//     Term 29 (AT2000-0250)/CC Inputs/Current actual value Ch.12 <-> Data Pointer/CurrentActualValues[11]
//     Term 29 (AT2000-0250)/CC Inputs/Current actual value Ch.13 <-> Data Pointer/CurrentActualValues[12]
//     Term 29 (AT2000-0250)/CC Inputs/Current actual value Ch.14 <-> Data Pointer/CurrentActualValues[13]
//     Term 29 (AT2000-0250)/CC Inputs/Current actual value Ch.15 <-> Data Pointer/CurrentActualValues[14]
//     Term 29 (AT2000-0250)/CC Inputs/Current actual value Ch.2 <-> Data Pointer/CurrentActualValues[1]
//     Term 29 (AT2000-0250)/CC Inputs/Current actual value Ch.3 <-> Data Pointer/CurrentActualValues[2]
//     Term 29 (AT2000-0250)/CC Inputs/Current actual value Ch.4 <-> Data Pointer/CurrentActualValues[3]
//     Term 29 (AT2000-0250)/CC Inputs/Current actual value Ch.5 <-> Data Pointer/CurrentActualValues[4]
//     Term 29 (AT2000-0250)/CC Inputs/Current actual value Ch.6 <-> Data Pointer/CurrentActualValues[5]
//     Term 29 (AT2000-0250)/CC Inputs/Current actual value Ch.7 <-> Data Pointer/CurrentActualValues[6]
//     Term 29 (AT2000-0250)/CC Inputs/Current actual value Ch.8 <-> Data Pointer/CurrentActualValues[7]
//     Term 29 (AT2000-0250)/CC Inputs/Current actual value Ch.9 <-> Data Pointer/CurrentActualValues[8]
//     Term 29 (AT2000-0250)/CC Inputs/Status <-> Data Pointer/Status
//     Term 29 (AT2000-0250)/CC Outputs/Control <-> Data Pointer/Control
//     Term 29 (AT2000-0250)/CC Outputs/Current setpoint value Ch.1 <-> Data Pointer/CurrentSetpointValues[0]
//     Term 29 (AT2000-0250)/CC Outputs/Current setpoint value Ch.10 <-> Data Pointer/CurrentSetpointValues[9]
//     Term 29 (AT2000-0250)/CC Outputs/Current setpoint value Ch.11 <-> Data Pointer/CurrentSetpointValues[10]
//     Term 29 (AT2000-0250)/CC Outputs/Current setpoint value Ch.12 <-> Data Pointer/CurrentSetpointValues[11]
//     Term 29 (AT2000-0250)/CC Outputs/Current setpoint value Ch.13 <-> Data Pointer/CurrentSetpointValues[12]
//     Term 29 (AT2000-0250)/CC Outputs/Current setpoint value Ch.14 <-> Data Pointer/CurrentSetpointValues[13]
//     Term 29 (AT2000-0250)/CC Outputs/Current setpoint value Ch.15 <-> Data Pointer/CurrentSetpointValues[14]
//     Term 29 (AT2000-0250)/CC Outputs/Current setpoint value Ch.2 <-> Data Pointer/CurrentSetpointValues[1]
//     Term 29 (AT2000-0250)/CC Outputs/Current setpoint value Ch.3 <-> Data Pointer/CurrentSetpointValues[2]
//     Term 29 (AT2000-0250)/CC Outputs/Current setpoint value Ch.4 <-> Data Pointer/CurrentSetpointValues[3]
//     Term 29 (AT2000-0250)/CC Outputs/Current setpoint value Ch.5 <-> Data Pointer/CurrentSetpointValues[4]
//     Term 29 (AT2000-0250)/CC Outputs/Current setpoint value Ch.6 <-> Data Pointer/CurrentSetpointValues[5]
//     Term 29 (AT2000-0250)/CC Outputs/Current setpoint value Ch.7 <-> Data Pointer/CurrentSetpointValues[6]
//     Term 29 (AT2000-0250)/CC Outputs/Current setpoint value Ch.8 <-> Data Pointer/CurrentSetpointValues[7]
//     Term 29 (AT2000-0250)/CC Outputs/Current setpoint value Ch.9 <-> Data Pointer/CurrentSetpointValues[8]
//     Term 29 (AT2000-0250)/Term 30 (AT2000-5250)/FB Inputs/Value Channel 01 <-> Data Pointer/RawPositionValues[0]
//     Term 29 (AT2000-0250)/Term 30 (AT2000-5250)/FB Inputs/Value Channel 02 <-> Data Pointer/RawPositionValues[1]
//     Term 29 (AT2000-0250)/Term 30 (AT2000-5250)/FB Inputs/Value Channel 03 <-> Data Pointer/RawPositionValues[2]
//     Term 29 (AT2000-0250)/Term 30 (AT2000-5250)/FB Inputs/Value Channel 04 <-> Data Pointer/RawPositionValues[3]
//     Term 29 (AT2000-0250)/Term 30 (AT2000-5250)/FB Inputs/Value Channel 05 <-> Data Pointer/RawPositionValues[4]
//     Term 29 (AT2000-0250)/Term 30 (AT2000-5250)/FB Inputs/Value Channel 06 <-> Data Pointer/RawPositionValues[5]
//     Term 29 (AT2000-0250)/Term 30 (AT2000-5250)/FB Inputs/Value Channel 07 <-> Data Pointer/RawPositionValues[6]
//     Term 29 (AT2000-0250)/Term 30 (AT2000-5250)/FB Inputs/Value Channel 08 <-> Data Pointer/RawPositionValues[7]
//     Term 29 (AT2000-0250)/Term 30 (AT2000-5250)/FB Inputs/Value Channel 09 <-> Data Pointer/RawPositionValues[8]
//     Term 29 (AT2000-0250)/Term 30 (AT2000-5250)/FB Inputs/Value Channel 10 <-> Data Pointer/RawPositionValues[9]
//     Term 29 (AT2000-0250)/Term 30 (AT2000-5250)/FB Inputs/Value Channel 11 <-> Data Pointer/RawPositionValues[10]
//     Term 29 (AT2000-0250)/Term 30 (AT2000-5250)/FB Inputs/Value Channel 12 <-> Data Pointer/RawPositionValues[11]
//     Term 29 (AT2000-0250)/Term 30 (AT2000-5250)/FB Inputs/Value Channel 13 <-> Data Pointer/RawPositionValues[12]
//     Term 29 (AT2000-0250)/Term 30 (AT2000-5250)/FB Inputs/Value Channel 14 <-> Data Pointer/RawPositionValues[13]
//     Term 29 (AT2000-0250)/Term 30 (AT2000-5250)/FB Inputs/Value Channel 15 <-> Data Pointer/RawPositionValues[14]
//     Term 29 (AT2000-0250)/Term 30 (AT2000-5250)/FB Inputs/Value Channel 16 <-> Data Pointer/RawPositionValues[15]
//     Term 29 (AT2000-0250)/Term 30 (AT2000-5250)/FB Inputs/Value Channel 17 <-> Data Pointer/RawPositionValues[16]
//     Term 29 (AT2000-0250)/Term 30 (AT2000-5250)/FB Inputs/Value Channel 18 <-> Data Pointer/RawPositionValues[17]
//     Term 29 (AT2000-0250)/Term 30 (AT2000-5250)/FB Inputs/Value Channel 19 <-> Data Pointer/RawPositionValues[18]
//     Term 29 (AT2000-0250)/Term 30 (AT2000-5250)/FB Inputs/Value Channel 20 <-> Data Pointer/RawPositionValues[19]
//     Term 29 (AT2000-0250)/Term 30 (AT2000-5250)/FB Inputs/Value Channel 21 <-> Data Pointer/RawPositionValues[20]
//     Term 29 (AT2000-0250)/Term 30 (AT2000-5250)/FB Inputs/Value Channel 22 <-> Data Pointer/RawPositionValues[21]
//     Term 29 (AT2000-0250)/Term 30 (AT2000-5250)/FB Inputs/Value Channel 23 <-> Data Pointer/RawPositionValues[22]
//     Term 29 (AT2000-0250)/Term 30 (AT2000-5250)/FB Inputs/Value Channel 24 <-> Data Pointer/RawPositionValues[23]
//     Term 29 (AT2000-0250)/Term 30 (AT2000-5250)/FB Inputs/Value Channel 25 <-> Data Pointer/RawPositionValues[24]
//     Term 29 (AT2000-0250)/Term 30 (AT2000-5250)/FB Inputs/Value Channel 26 <-> Data Pointer/RawPositionValues[25]
//     Term 29 (AT2000-0250)/Term 30 (AT2000-5250)/FB Inputs/Value Channel 27 <-> Data Pointer/RawPositionValues[26]
//     Term 29 (AT2000-0250)/Term 30 (AT2000-5250)/FB Inputs/Value Channel 28 <-> Data Pointer/RawPositionValues[27]
//     Term 29 (AT2000-0250)/Term 30 (AT2000-5250)/FB Inputs/Value Channel 29 <-> Data Pointer/RawPositionValues[28]
//     Term 29 (AT2000-0250)/Term 30 (AT2000-5250)/FB Inputs/Value Channel 30 <-> Data Pointer/RawPositionValues[29]
//     Term 29 (AT2000-0250)/Term 30 (AT2000-5250)/FB Inputs/Value Channel 31 <-> Data Pointer/RawPositionValues[30]
//     Term 29 (AT2000-0250)/Term 30 (AT2000-5250)/FB Inputs/Value Channel 32 <-> Data Pointer/RawPositionValues[31]
//   Device 4 (EtherCAT) <-> TcCOM Objects/Object7 (CTcIoXtsDrv)/XTS Module Adapter_Obj15 (AT2050_X500)
//     Term 31 (AT2050-0500)/CC Inputs/Current actual value Ch.1 <-> Data Pointer/CurrentActualValues[0]
//     Term 31 (AT2050-0500)/CC Inputs/Current actual value Ch.10 <-> Data Pointer/CurrentActualValues[9]
//     Term 31 (AT2050-0500)/CC Inputs/Current actual value Ch.11 <-> Data Pointer/CurrentActualValues[10]
//     Term 31 (AT2050-0500)/CC Inputs/Current actual value Ch.12 <-> Data Pointer/CurrentActualValues[11]
//     Term 31 (AT2050-0500)/CC Inputs/Current actual value Ch.13 <-> Data Pointer/CurrentActualValues[12]
//     Term 31 (AT2050-0500)/CC Inputs/Current actual value Ch.14 <-> Data Pointer/CurrentActualValues[13]
//     Term 31 (AT2050-0500)/CC Inputs/Current actual value Ch.15 <-> Data Pointer/CurrentActualValues[14]
//     Term 31 (AT2050-0500)/CC Inputs/Current actual value Ch.2 <-> Data Pointer/CurrentActualValues[1]
//     Term 31 (AT2050-0500)/CC Inputs/Current actual value Ch.3 <-> Data Pointer/CurrentActualValues[2]
//     Term 31 (AT2050-0500)/CC Inputs/Current actual value Ch.4 <-> Data Pointer/CurrentActualValues[3]
//     Term 31 (AT2050-0500)/CC Inputs/Current actual value Ch.5 <-> Data Pointer/CurrentActualValues[4]
//     Term 31 (AT2050-0500)/CC Inputs/Current actual value Ch.6 <-> Data Pointer/CurrentActualValues[5]
//     Term 31 (AT2050-0500)/CC Inputs/Current actual value Ch.7 <-> Data Pointer/CurrentActualValues[6]
//     Term 31 (AT2050-0500)/CC Inputs/Current actual value Ch.8 <-> Data Pointer/CurrentActualValues[7]
//     Term 31 (AT2050-0500)/CC Inputs/Current actual value Ch.9 <-> Data Pointer/CurrentActualValues[8]
//     Term 31 (AT2050-0500)/CC Inputs/Status <-> Data Pointer/Status
//     Term 31 (AT2050-0500)/CC Outputs/Control <-> Data Pointer/Control
//     Term 31 (AT2050-0500)/CC Outputs/Current setpoint value Ch.1 <-> Data Pointer/CurrentSetpointValues[0]
//     Term 31 (AT2050-0500)/CC Outputs/Current setpoint value Ch.10 <-> Data Pointer/CurrentSetpointValues[9]
//     Term 31 (AT2050-0500)/CC Outputs/Current setpoint value Ch.11 <-> Data Pointer/CurrentSetpointValues[10]
//     Term 31 (AT2050-0500)/CC Outputs/Current setpoint value Ch.12 <-> Data Pointer/CurrentSetpointValues[11]
//     Term 31 (AT2050-0500)/CC Outputs/Current setpoint value Ch.13 <-> Data Pointer/CurrentSetpointValues[12]
//     Term 31 (AT2050-0500)/CC Outputs/Current setpoint value Ch.14 <-> Data Pointer/CurrentSetpointValues[13]
//     Term 31 (AT2050-0500)/CC Outputs/Current setpoint value Ch.15 <-> Data Pointer/CurrentSetpointValues[14]
//     Term 31 (AT2050-0500)/CC Outputs/Current setpoint value Ch.2 <-> Data Pointer/CurrentSetpointValues[1]
//     Term 31 (AT2050-0500)/CC Outputs/Current setpoint value Ch.3 <-> Data Pointer/CurrentSetpointValues[2]
//     Term 31 (AT2050-0500)/CC Outputs/Current setpoint value Ch.4 <-> Data Pointer/CurrentSetpointValues[3]
//     Term 31 (AT2050-0500)/CC Outputs/Current setpoint value Ch.5 <-> Data Pointer/CurrentSetpointValues[4]
//     Term 31 (AT2050-0500)/CC Outputs/Current setpoint value Ch.6 <-> Data Pointer/CurrentSetpointValues[5]
//     Term 31 (AT2050-0500)/CC Outputs/Current setpoint value Ch.7 <-> Data Pointer/CurrentSetpointValues[6]
//     Term 31 (AT2050-0500)/CC Outputs/Current setpoint value Ch.8 <-> Data Pointer/CurrentSetpointValues[7]
//     Term 31 (AT2050-0500)/CC Outputs/Current setpoint value Ch.9 <-> Data Pointer/CurrentSetpointValues[8]
//     Term 31 (AT2050-0500)/Term 32 (AT2050-5500)/FB Inputs/Value Channel 01 <-> Data Pointer/RawPositionValues[0]
//     Term 31 (AT2050-0500)/Term 32 (AT2050-5500)/FB Inputs/Value Channel 02 <-> Data Pointer/RawPositionValues[1]
//     Term 31 (AT2050-0500)/Term 32 (AT2050-5500)/FB Inputs/Value Channel 03 <-> Data Pointer/RawPositionValues[2]
//     Term 31 (AT2050-0500)/Term 32 (AT2050-5500)/FB Inputs/Value Channel 04 <-> Data Pointer/RawPositionValues[3]
//     Term 31 (AT2050-0500)/Term 32 (AT2050-5500)/FB Inputs/Value Channel 05 <-> Data Pointer/RawPositionValues[4]
//     Term 31 (AT2050-0500)/Term 32 (AT2050-5500)/FB Inputs/Value Channel 06 <-> Data Pointer/RawPositionValues[5]
//     Term 31 (AT2050-0500)/Term 32 (AT2050-5500)/FB Inputs/Value Channel 07 <-> Data Pointer/RawPositionValues[6]
//     Term 31 (AT2050-0500)/Term 32 (AT2050-5500)/FB Inputs/Value Channel 08 <-> Data Pointer/RawPositionValues[7]
//     Term 31 (AT2050-0500)/Term 32 (AT2050-5500)/FB Inputs/Value Channel 09 <-> Data Pointer/RawPositionValues[8]
//     Term 31 (AT2050-0500)/Term 32 (AT2050-5500)/FB Inputs/Value Channel 10 <-> Data Pointer/RawPositionValues[9]
//     Term 31 (AT2050-0500)/Term 32 (AT2050-5500)/FB Inputs/Value Channel 11 <-> Data Pointer/RawPositionValues[10]
//     Term 31 (AT2050-0500)/Term 32 (AT2050-5500)/FB Inputs/Value Channel 12 <-> Data Pointer/RawPositionValues[11]
//     Term 31 (AT2050-0500)/Term 32 (AT2050-5500)/FB Inputs/Value Channel 13 <-> Data Pointer/RawPositionValues[12]
//     Term 31 (AT2050-0500)/Term 32 (AT2050-5500)/FB Inputs/Value Channel 14 <-> Data Pointer/RawPositionValues[13]
//     Term 31 (AT2050-0500)/Term 32 (AT2050-5500)/FB Inputs/Value Channel 15 <-> Data Pointer/RawPositionValues[14]
//     Term 31 (AT2050-0500)/Term 32 (AT2050-5500)/FB Inputs/Value Channel 16 <-> Data Pointer/RawPositionValues[15]
//     Term 31 (AT2050-0500)/Term 32 (AT2050-5500)/FB Inputs/Value Channel 17 <-> Data Pointer/RawPositionValues[16]
//     Term 31 (AT2050-0500)/Term 32 (AT2050-5500)/FB Inputs/Value Channel 18 <-> Data Pointer/RawPositionValues[17]
//     Term 31 (AT2050-0500)/Term 32 (AT2050-5500)/FB Inputs/Value Channel 19 <-> Data Pointer/RawPositionValues[18]
//     Term 31 (AT2050-0500)/Term 32 (AT2050-5500)/FB Inputs/Value Channel 20 <-> Data Pointer/RawPositionValues[19]
//     Term 31 (AT2050-0500)/Term 32 (AT2050-5500)/FB Inputs/Value Channel 21 <-> Data Pointer/RawPositionValues[20]
//     Term 31 (AT2050-0500)/Term 32 (AT2050-5500)/FB Inputs/Value Channel 22 <-> Data Pointer/RawPositionValues[21]
//     Term 31 (AT2050-0500)/Term 32 (AT2050-5500)/FB Inputs/Value Channel 23 <-> Data Pointer/RawPositionValues[22]
//     Term 31 (AT2050-0500)/Term 32 (AT2050-5500)/FB Inputs/Value Channel 24 <-> Data Pointer/RawPositionValues[23]
//     Term 31 (AT2050-0500)/Term 32 (AT2050-5500)/FB Inputs/Value Channel 25 <-> Data Pointer/RawPositionValues[24]
//     Term 31 (AT2050-0500)/Term 32 (AT2050-5500)/FB Inputs/Value Channel 26 <-> Data Pointer/RawPositionValues[25]
//     Term 31 (AT2050-0500)/Term 32 (AT2050-5500)/FB Inputs/Value Channel 27 <-> Data Pointer/RawPositionValues[26]
//     Term 31 (AT2050-0500)/Term 32 (AT2050-5500)/FB Inputs/Value Channel 28 <-> Data Pointer/RawPositionValues[27]
//     Term 31 (AT2050-0500)/Term 32 (AT2050-5500)/FB Inputs/Value Channel 29 <-> Data Pointer/RawPositionValues[28]
//     Term 31 (AT2050-0500)/Term 32 (AT2050-5500)/FB Inputs/Value Channel 30 <-> Data Pointer/RawPositionValues[29]
//     Term 31 (AT2050-0500)/Term 32 (AT2050-5500)/FB Inputs/Value Channel 31 <-> Data Pointer/RawPositionValues[30]
//     Term 31 (AT2050-0500)/Term 32 (AT2050-5500)/FB Inputs/Value Channel 32 <-> Data Pointer/RawPositionValues[31]
//   Device 4 (EtherCAT) <-> TcCOM Objects/Object7 (CTcIoXtsDrv)/XTS Module Adapter_Obj16 (AT2050_X501)
//     Term 33 (AT2050-0501)/CC Inputs/Current actual value Ch.1 <-> Data Pointer/CurrentActualValues[0]
//     Term 33 (AT2050-0501)/CC Inputs/Current actual value Ch.10 <-> Data Pointer/CurrentActualValues[9]
//     Term 33 (AT2050-0501)/CC Inputs/Current actual value Ch.11 <-> Data Pointer/CurrentActualValues[10]
//     Term 33 (AT2050-0501)/CC Inputs/Current actual value Ch.12 <-> Data Pointer/CurrentActualValues[11]
//     Term 33 (AT2050-0501)/CC Inputs/Current actual value Ch.13 <-> Data Pointer/CurrentActualValues[12]
//     Term 33 (AT2050-0501)/CC Inputs/Current actual value Ch.14 <-> Data Pointer/CurrentActualValues[13]
//     Term 33 (AT2050-0501)/CC Inputs/Current actual value Ch.15 <-> Data Pointer/CurrentActualValues[14]
//     Term 33 (AT2050-0501)/CC Inputs/Current actual value Ch.2 <-> Data Pointer/CurrentActualValues[1]
//     Term 33 (AT2050-0501)/CC Inputs/Current actual value Ch.3 <-> Data Pointer/CurrentActualValues[2]
//     Term 33 (AT2050-0501)/CC Inputs/Current actual value Ch.4 <-> Data Pointer/CurrentActualValues[3]
//     Term 33 (AT2050-0501)/CC Inputs/Current actual value Ch.5 <-> Data Pointer/CurrentActualValues[4]
//     Term 33 (AT2050-0501)/CC Inputs/Current actual value Ch.6 <-> Data Pointer/CurrentActualValues[5]
//     Term 33 (AT2050-0501)/CC Inputs/Current actual value Ch.7 <-> Data Pointer/CurrentActualValues[6]
//     Term 33 (AT2050-0501)/CC Inputs/Current actual value Ch.8 <-> Data Pointer/CurrentActualValues[7]
//     Term 33 (AT2050-0501)/CC Inputs/Current actual value Ch.9 <-> Data Pointer/CurrentActualValues[8]
//     Term 33 (AT2050-0501)/CC Inputs/Status <-> Data Pointer/Status
//     Term 33 (AT2050-0501)/CC Outputs/Control <-> Data Pointer/Control
//     Term 33 (AT2050-0501)/CC Outputs/Current setpoint value Ch.1 <-> Data Pointer/CurrentSetpointValues[0]
//     Term 33 (AT2050-0501)/CC Outputs/Current setpoint value Ch.10 <-> Data Pointer/CurrentSetpointValues[9]
//     Term 33 (AT2050-0501)/CC Outputs/Current setpoint value Ch.11 <-> Data Pointer/CurrentSetpointValues[10]
//     Term 33 (AT2050-0501)/CC Outputs/Current setpoint value Ch.12 <-> Data Pointer/CurrentSetpointValues[11]
//     Term 33 (AT2050-0501)/CC Outputs/Current setpoint value Ch.13 <-> Data Pointer/CurrentSetpointValues[12]
//     Term 33 (AT2050-0501)/CC Outputs/Current setpoint value Ch.14 <-> Data Pointer/CurrentSetpointValues[13]
//     Term 33 (AT2050-0501)/CC Outputs/Current setpoint value Ch.15 <-> Data Pointer/CurrentSetpointValues[14]
//     Term 33 (AT2050-0501)/CC Outputs/Current setpoint value Ch.2 <-> Data Pointer/CurrentSetpointValues[1]
//     Term 33 (AT2050-0501)/CC Outputs/Current setpoint value Ch.3 <-> Data Pointer/CurrentSetpointValues[2]
//     Term 33 (AT2050-0501)/CC Outputs/Current setpoint value Ch.4 <-> Data Pointer/CurrentSetpointValues[3]
//     Term 33 (AT2050-0501)/CC Outputs/Current setpoint value Ch.5 <-> Data Pointer/CurrentSetpointValues[4]
//     Term 33 (AT2050-0501)/CC Outputs/Current setpoint value Ch.6 <-> Data Pointer/CurrentSetpointValues[5]
//     Term 33 (AT2050-0501)/CC Outputs/Current setpoint value Ch.7 <-> Data Pointer/CurrentSetpointValues[6]
//     Term 33 (AT2050-0501)/CC Outputs/Current setpoint value Ch.8 <-> Data Pointer/CurrentSetpointValues[7]
//     Term 33 (AT2050-0501)/CC Outputs/Current setpoint value Ch.9 <-> Data Pointer/CurrentSetpointValues[8]
//     Term 33 (AT2050-0501)/Term 34 (AT2050-5501)/FB Inputs/Value Channel 01 <-> Data Pointer/RawPositionValues[0]
//     Term 33 (AT2050-0501)/Term 34 (AT2050-5501)/FB Inputs/Value Channel 02 <-> Data Pointer/RawPositionValues[1]
//     Term 33 (AT2050-0501)/Term 34 (AT2050-5501)/FB Inputs/Value Channel 03 <-> Data Pointer/RawPositionValues[2]
//     Term 33 (AT2050-0501)/Term 34 (AT2050-5501)/FB Inputs/Value Channel 04 <-> Data Pointer/RawPositionValues[3]
//     Term 33 (AT2050-0501)/Term 34 (AT2050-5501)/FB Inputs/Value Channel 05 <-> Data Pointer/RawPositionValues[4]
//     Term 33 (AT2050-0501)/Term 34 (AT2050-5501)/FB Inputs/Value Channel 06 <-> Data Pointer/RawPositionValues[5]
//     Term 33 (AT2050-0501)/Term 34 (AT2050-5501)/FB Inputs/Value Channel 07 <-> Data Pointer/RawPositionValues[6]
//     Term 33 (AT2050-0501)/Term 34 (AT2050-5501)/FB Inputs/Value Channel 08 <-> Data Pointer/RawPositionValues[7]
//     Term 33 (AT2050-0501)/Term 34 (AT2050-5501)/FB Inputs/Value Channel 09 <-> Data Pointer/RawPositionValues[8]
//     Term 33 (AT2050-0501)/Term 34 (AT2050-5501)/FB Inputs/Value Channel 10 <-> Data Pointer/RawPositionValues[9]
//     Term 33 (AT2050-0501)/Term 34 (AT2050-5501)/FB Inputs/Value Channel 11 <-> Data Pointer/RawPositionValues[10]
//     Term 33 (AT2050-0501)/Term 34 (AT2050-5501)/FB Inputs/Value Channel 12 <-> Data Pointer/RawPositionValues[11]
//     Term 33 (AT2050-0501)/Term 34 (AT2050-5501)/FB Inputs/Value Channel 13 <-> Data Pointer/RawPositionValues[12]
//     Term 33 (AT2050-0501)/Term 34 (AT2050-5501)/FB Inputs/Value Channel 14 <-> Data Pointer/RawPositionValues[13]
//     Term 33 (AT2050-0501)/Term 34 (AT2050-5501)/FB Inputs/Value Channel 15 <-> Data Pointer/RawPositionValues[14]
//     Term 33 (AT2050-0501)/Term 34 (AT2050-5501)/FB Inputs/Value Channel 16 <-> Data Pointer/RawPositionValues[15]
//     Term 33 (AT2050-0501)/Term 34 (AT2050-5501)/FB Inputs/Value Channel 17 <-> Data Pointer/RawPositionValues[16]
//     Term 33 (AT2050-0501)/Term 34 (AT2050-5501)/FB Inputs/Value Channel 18 <-> Data Pointer/RawPositionValues[17]
//     Term 33 (AT2050-0501)/Term 34 (AT2050-5501)/FB Inputs/Value Channel 19 <-> Data Pointer/RawPositionValues[18]
//     Term 33 (AT2050-0501)/Term 34 (AT2050-5501)/FB Inputs/Value Channel 20 <-> Data Pointer/RawPositionValues[19]
//     Term 33 (AT2050-0501)/Term 34 (AT2050-5501)/FB Inputs/Value Channel 21 <-> Data Pointer/RawPositionValues[20]
//     Term 33 (AT2050-0501)/Term 34 (AT2050-5501)/FB Inputs/Value Channel 22 <-> Data Pointer/RawPositionValues[21]
//     Term 33 (AT2050-0501)/Term 34 (AT2050-5501)/FB Inputs/Value Channel 23 <-> Data Pointer/RawPositionValues[22]
//     Term 33 (AT2050-0501)/Term 34 (AT2050-5501)/FB Inputs/Value Channel 24 <-> Data Pointer/RawPositionValues[23]
//     Term 33 (AT2050-0501)/Term 34 (AT2050-5501)/FB Inputs/Value Channel 25 <-> Data Pointer/RawPositionValues[24]
//     Term 33 (AT2050-0501)/Term 34 (AT2050-5501)/FB Inputs/Value Channel 26 <-> Data Pointer/RawPositionValues[25]
//     Term 33 (AT2050-0501)/Term 34 (AT2050-5501)/FB Inputs/Value Channel 27 <-> Data Pointer/RawPositionValues[26]
//     Term 33 (AT2050-0501)/Term 34 (AT2050-5501)/FB Inputs/Value Channel 28 <-> Data Pointer/RawPositionValues[27]
//     Term 33 (AT2050-0501)/Term 34 (AT2050-5501)/FB Inputs/Value Channel 29 <-> Data Pointer/RawPositionValues[28]
//     Term 33 (AT2050-0501)/Term 34 (AT2050-5501)/FB Inputs/Value Channel 30 <-> Data Pointer/RawPositionValues[29]
//     Term 33 (AT2050-0501)/Term 34 (AT2050-5501)/FB Inputs/Value Channel 31 <-> Data Pointer/RawPositionValues[30]
//     Term 33 (AT2050-0501)/Term 34 (AT2050-5501)/FB Inputs/Value Channel 32 <-> Data Pointer/RawPositionValues[31]
//   Device 4 (EtherCAT) <-> TcCOM Objects/Object7 (CTcIoXtsDrv)/XTS Module Adapter_Obj9 (AT2001_X250)
//     Term 19 (AT2001-0250)/CC Inputs/Current actual value Ch.1 <-> Data Pointer/CurrentActualValues[0]
//     Term 19 (AT2001-0250)/CC Inputs/Current actual value Ch.10 <-> Data Pointer/CurrentActualValues[9]
//     Term 19 (AT2001-0250)/CC Inputs/Current actual value Ch.11 <-> Data Pointer/CurrentActualValues[10]
//     Term 19 (AT2001-0250)/CC Inputs/Current actual value Ch.12 <-> Data Pointer/CurrentActualValues[11]
//     Term 19 (AT2001-0250)/CC Inputs/Current actual value Ch.13 <-> Data Pointer/CurrentActualValues[12]
//     Term 19 (AT2001-0250)/CC Inputs/Current actual value Ch.14 <-> Data Pointer/CurrentActualValues[13]
//     Term 19 (AT2001-0250)/CC Inputs/Current actual value Ch.15 <-> Data Pointer/CurrentActualValues[14]
//     Term 19 (AT2001-0250)/CC Inputs/Current actual value Ch.2 <-> Data Pointer/CurrentActualValues[1]
//     Term 19 (AT2001-0250)/CC Inputs/Current actual value Ch.3 <-> Data Pointer/CurrentActualValues[2]
//     Term 19 (AT2001-0250)/CC Inputs/Current actual value Ch.4 <-> Data Pointer/CurrentActualValues[3]
//     Term 19 (AT2001-0250)/CC Inputs/Current actual value Ch.5 <-> Data Pointer/CurrentActualValues[4]
//     Term 19 (AT2001-0250)/CC Inputs/Current actual value Ch.6 <-> Data Pointer/CurrentActualValues[5]
//     Term 19 (AT2001-0250)/CC Inputs/Current actual value Ch.7 <-> Data Pointer/CurrentActualValues[6]
//     Term 19 (AT2001-0250)/CC Inputs/Current actual value Ch.8 <-> Data Pointer/CurrentActualValues[7]
//     Term 19 (AT2001-0250)/CC Inputs/Current actual value Ch.9 <-> Data Pointer/CurrentActualValues[8]
//     Term 19 (AT2001-0250)/CC Inputs/Status <-> Data Pointer/Status
//     Term 19 (AT2001-0250)/CC Outputs/Control <-> Data Pointer/Control
//     Term 19 (AT2001-0250)/CC Outputs/Current setpoint value Ch.1 <-> Data Pointer/CurrentSetpointValues[0]
//     Term 19 (AT2001-0250)/CC Outputs/Current setpoint value Ch.10 <-> Data Pointer/CurrentSetpointValues[9]
//     Term 19 (AT2001-0250)/CC Outputs/Current setpoint value Ch.11 <-> Data Pointer/CurrentSetpointValues[10]
//     Term 19 (AT2001-0250)/CC Outputs/Current setpoint value Ch.12 <-> Data Pointer/CurrentSetpointValues[11]
//     Term 19 (AT2001-0250)/CC Outputs/Current setpoint value Ch.13 <-> Data Pointer/CurrentSetpointValues[12]
//     Term 19 (AT2001-0250)/CC Outputs/Current setpoint value Ch.14 <-> Data Pointer/CurrentSetpointValues[13]
//     Term 19 (AT2001-0250)/CC Outputs/Current setpoint value Ch.15 <-> Data Pointer/CurrentSetpointValues[14]
//     Term 19 (AT2001-0250)/CC Outputs/Current setpoint value Ch.2 <-> Data Pointer/CurrentSetpointValues[1]
//     Term 19 (AT2001-0250)/CC Outputs/Current setpoint value Ch.3 <-> Data Pointer/CurrentSetpointValues[2]
//     Term 19 (AT2001-0250)/CC Outputs/Current setpoint value Ch.4 <-> Data Pointer/CurrentSetpointValues[3]
//     Term 19 (AT2001-0250)/CC Outputs/Current setpoint value Ch.5 <-> Data Pointer/CurrentSetpointValues[4]
//     Term 19 (AT2001-0250)/CC Outputs/Current setpoint value Ch.6 <-> Data Pointer/CurrentSetpointValues[5]
//     Term 19 (AT2001-0250)/CC Outputs/Current setpoint value Ch.7 <-> Data Pointer/CurrentSetpointValues[6]
//     Term 19 (AT2001-0250)/CC Outputs/Current setpoint value Ch.8 <-> Data Pointer/CurrentSetpointValues[7]
//     Term 19 (AT2001-0250)/CC Outputs/Current setpoint value Ch.9 <-> Data Pointer/CurrentSetpointValues[8]
//     Term 19 (AT2001-0250)/Term 20 (AT2001-5250)/FB Inputs/Value Channel 01 <-> Data Pointer/RawPositionValues[0]
//     Term 19 (AT2001-0250)/Term 20 (AT2001-5250)/FB Inputs/Value Channel 02 <-> Data Pointer/RawPositionValues[1]
//     Term 19 (AT2001-0250)/Term 20 (AT2001-5250)/FB Inputs/Value Channel 03 <-> Data Pointer/RawPositionValues[2]
//     Term 19 (AT2001-0250)/Term 20 (AT2001-5250)/FB Inputs/Value Channel 04 <-> Data Pointer/RawPositionValues[3]
//     Term 19 (AT2001-0250)/Term 20 (AT2001-5250)/FB Inputs/Value Channel 05 <-> Data Pointer/RawPositionValues[4]
//     Term 19 (AT2001-0250)/Term 20 (AT2001-5250)/FB Inputs/Value Channel 06 <-> Data Pointer/RawPositionValues[5]
//     Term 19 (AT2001-0250)/Term 20 (AT2001-5250)/FB Inputs/Value Channel 07 <-> Data Pointer/RawPositionValues[6]
//     Term 19 (AT2001-0250)/Term 20 (AT2001-5250)/FB Inputs/Value Channel 08 <-> Data Pointer/RawPositionValues[7]
//     Term 19 (AT2001-0250)/Term 20 (AT2001-5250)/FB Inputs/Value Channel 09 <-> Data Pointer/RawPositionValues[8]
//     Term 19 (AT2001-0250)/Term 20 (AT2001-5250)/FB Inputs/Value Channel 10 <-> Data Pointer/RawPositionValues[9]
//     Term 19 (AT2001-0250)/Term 20 (AT2001-5250)/FB Inputs/Value Channel 11 <-> Data Pointer/RawPositionValues[10]
//     Term 19 (AT2001-0250)/Term 20 (AT2001-5250)/FB Inputs/Value Channel 12 <-> Data Pointer/RawPositionValues[11]
//     Term 19 (AT2001-0250)/Term 20 (AT2001-5250)/FB Inputs/Value Channel 13 <-> Data Pointer/RawPositionValues[12]
//     Term 19 (AT2001-0250)/Term 20 (AT2001-5250)/FB Inputs/Value Channel 14 <-> Data Pointer/RawPositionValues[13]
//     Term 19 (AT2001-0250)/Term 20 (AT2001-5250)/FB Inputs/Value Channel 15 <-> Data Pointer/RawPositionValues[14]
//     Term 19 (AT2001-0250)/Term 20 (AT2001-5250)/FB Inputs/Value Channel 16 <-> Data Pointer/RawPositionValues[15]
//     Term 19 (AT2001-0250)/Term 20 (AT2001-5250)/FB Inputs/Value Channel 17 <-> Data Pointer/RawPositionValues[16]
//     Term 19 (AT2001-0250)/Term 20 (AT2001-5250)/FB Inputs/Value Channel 18 <-> Data Pointer/RawPositionValues[17]
//     Term 19 (AT2001-0250)/Term 20 (AT2001-5250)/FB Inputs/Value Channel 19 <-> Data Pointer/RawPositionValues[18]
//     Term 19 (AT2001-0250)/Term 20 (AT2001-5250)/FB Inputs/Value Channel 20 <-> Data Pointer/RawPositionValues[19]
//     Term 19 (AT2001-0250)/Term 20 (AT2001-5250)/FB Inputs/Value Channel 21 <-> Data Pointer/RawPositionValues[20]
//     Term 19 (AT2001-0250)/Term 20 (AT2001-5250)/FB Inputs/Value Channel 22 <-> Data Pointer/RawPositionValues[21]
//     Term 19 (AT2001-0250)/Term 20 (AT2001-5250)/FB Inputs/Value Channel 23 <-> Data Pointer/RawPositionValues[22]
//     Term 19 (AT2001-0250)/Term 20 (AT2001-5250)/FB Inputs/Value Channel 24 <-> Data Pointer/RawPositionValues[23]
//     Term 19 (AT2001-0250)/Term 20 (AT2001-5250)/FB Inputs/Value Channel 25 <-> Data Pointer/RawPositionValues[24]
//     Term 19 (AT2001-0250)/Term 20 (AT2001-5250)/FB Inputs/Value Channel 26 <-> Data Pointer/RawPositionValues[25]
//     Term 19 (AT2001-0250)/Term 20 (AT2001-5250)/FB Inputs/Value Channel 27 <-> Data Pointer/RawPositionValues[26]
//     Term 19 (AT2001-0250)/Term 20 (AT2001-5250)/FB Inputs/Value Channel 28 <-> Data Pointer/RawPositionValues[27]
//     Term 19 (AT2001-0250)/Term 20 (AT2001-5250)/FB Inputs/Value Channel 29 <-> Data Pointer/RawPositionValues[28]
//     Term 19 (AT2001-0250)/Term 20 (AT2001-5250)/FB Inputs/Value Channel 30 <-> Data Pointer/RawPositionValues[29]
//     Term 19 (AT2001-0250)/Term 20 (AT2001-5250)/FB Inputs/Value Channel 31 <-> Data Pointer/RawPositionValues[30]
//     Term 19 (AT2001-0250)/Term 20 (AT2001-5250)/FB Inputs/Value Channel 32 <-> Data Pointer/RawPositionValues[31]
//   NC Task SAF/Axes/Axis 1 <-> TcCOM Objects/Object7 (CTcIoXtsDrv)/Mover 1_Obj17 (CMover)
//     SoftDrive 1_Obj1 (CTcSoftDrive)/Data Pointer/InputPointer1 <-> Inputs/SoftDriveInput
//     SoftDrive 1_Obj1 (CTcSoftDrive)/Data Pointer/OutputPointer1 <-> Outputs/SoftDriveOutput
//   NC Task SAF/Axes/Axis 2 <-> TcCOM Objects/Object7 (CTcIoXtsDrv)/Mover 2_Obj18 (CMover)
//     SoftDrive 2_Obj1 (CTcSoftDrive)/Data Pointer/InputPointer1 <-> Inputs/SoftDriveInput
//     SoftDrive 2_Obj1 (CTcSoftDrive)/Data Pointer/OutputPointer1 <-> Outputs/SoftDriveOutput
//   NC Task SAF/Axes/Axis 3 <-> TcCOM Objects/Object7 (CTcIoXtsDrv)/Mover 3_Obj19 (CMover)
//     SoftDrive 3_Obj1 (CTcSoftDrive)/Data Pointer/InputPointer1 <-> Inputs/SoftDriveInput
//     SoftDrive 3_Obj1 (CTcSoftDrive)/Data Pointer/OutputPointer1 <-> Outputs/SoftDriveOutput
//   NC Task SAF/Axes/Axis 4 <-> TcCOM Objects/Object7 (CTcIoXtsDrv)/Mover 4_Obj20 (CMover)
//     SoftDrive 4_Obj1 (CTcSoftDrive)/Data Pointer/InputPointer1 <-> Inputs/SoftDriveInput
//     SoftDrive 4_Obj1 (CTcSoftDrive)/Data Pointer/OutputPointer1 <-> Outputs/SoftDriveOutput
//   NC Task SAF/Axes/Axis 5 <-> TcCOM Objects/Object7 (CTcIoXtsDrv)/Mover 5_Obj21 (CMover)
//     SoftDrive 5_Obj1 (CTcSoftDrive)/Data Pointer/InputPointer1 <-> Inputs/SoftDriveInput
//     SoftDrive 5_Obj1 (CTcSoftDrive)/Data Pointer/OutputPointer1 <-> Outputs/SoftDriveOutput
//   NC Task SAF/Axes/Axis 6 <-> TcCOM Objects/Object7 (CTcIoXtsDrv)/Mover 6_Obj22 (CMover)
//     SoftDrive 6_Obj1 (CTcSoftDrive)/Data Pointer/InputPointer1 <-> Inputs/SoftDriveInput
//     SoftDrive 6_Obj1 (CTcSoftDrive)/Data Pointer/OutputPointer1 <-> Outputs/SoftDriveOutput
//   141114mi5XTSPLC/141114mi5XTSPLC Instance <-> NC Task SAF/Axes/Axis 1
//     PlcTask Inputs/GVL.ax[1].NcToPlc <-> Outputs/ToPlc
//     PlcTask Outputs/GVL.ax[1].PlcToNc <-> Inputs/FromPlc
//   141114mi5XTSPLC/141114mi5XTSPLC Instance <-> NC Task SAF/Axes/Axis 2
//     PlcTask Inputs/GVL.ax[2].NcToPlc <-> Outputs/ToPlc
//     PlcTask Outputs/GVL.ax[2].PlcToNc <-> Inputs/FromPlc
//   141114mi5XTSPLC/141114mi5XTSPLC Instance <-> NC Task SAF/Axes/Axis 3
//     PlcTask Inputs/GVL.ax[3].NcToPlc <-> Outputs/ToPlc
//     PlcTask Outputs/GVL.ax[3].PlcToNc <-> Inputs/FromPlc
//   141114mi5XTSPLC/141114mi5XTSPLC Instance <-> NC Task SAF/Axes/Axis 4
//     PlcTask Inputs/GVL.ax[4].NcToPlc <-> Outputs/ToPlc
//     PlcTask Outputs/GVL.ax[4].PlcToNc <-> Inputs/FromPlc
//   141114mi5XTSPLC/141114mi5XTSPLC Instance <-> NC Task SAF/Axes/Axis 5
//     PlcTask Inputs/GVL.ax[5].NcToPlc <-> Outputs/ToPlc
//     PlcTask Outputs/GVL.ax[5].PlcToNc <-> Inputs/FromPlc
//   141114mi5XTSPLC/141114mi5XTSPLC Instance <-> NC Task SAF/Axes/Axis 6
//     PlcTask Inputs/GVL.ax[6].NcToPlc <-> Outputs/ToPlc
//     PlcTask Outputs/GVL.ax[6].PlcToNc <-> Inputs/FromPlc
//   141114mi5XTSPLC/141114mi5XTSPLC Instance <-> NC Task SAF/Axes/Grp 1
//     PlcTask Inputs/GVL.grp[1].NcToPlc <-> Outputs/ToPlc
//     PlcTask Outputs/GVL.grp[1].PlcToNc <-> Inputs/FromPlc
//   141114mi5XTSPLC/141114mi5XTSPLC Instance <-> NC Task SAF/Axes/Grp 2
//     PlcTask Inputs/GVL.grp[2].NcToPlc <-> Outputs/ToPlc
//     PlcTask Outputs/GVL.grp[2].PlcToNc <-> Inputs/FromPlc
//   141114mi5XTSPLC/141114mi5XTSPLC Instance <-> NC Task SAF/Axes/Grp 3
//     PlcTask Inputs/GVL.grp[3].NcToPlc <-> Outputs/ToPlc
//     PlcTask Outputs/GVL.grp[3].PlcToNc <-> Inputs/FromPlc
//   141114mi5XTSPLC/141114mi5XTSPLC Instance <-> TcCOM Objects/CA Group_Obj3 (CA Group)
//     PlcTask Inputs/GVL.CAgrp.NcToPlc <-> Group Outputs/ToPLC
//     PlcTask Outputs/GVL.CAgrp.PlcToNc <-> Group Inputs/FromPLC
//   XTS Task <-> Device 3 (EtherCAT)
//     Inputs/Init_Strang1 <-> Inputs/DevState
//   XTS Task <-> Device 4 (EtherCAT)
//     Inputs/Init_Strang2 <-> Inputs/DevState

CONFIGURATION _141114mi5XTSPLC
    RESOURCE PLC ON TwinCAT3
        TASK PlcTask(INTERVAL := T#250us, PRIORITY := 1);
        TASK SimuTask(INTERVAL := T#10ms, PRIORITY := 2);
        PROGRAM OPC_Client WITH PlcTask : OPC_Client;
        PROGRAM Powerall WITH PlcTask : Powerall;
        PROGRAM MAIN WITH PlcTask : MAIN;
        PROGRAM MAIN_simu WITH SimuTask : MAIN_simu;
    END_RESOURCE
END_CONFIGURATION

// ---- DUTs/industrialPhysics/MNG_APPLICATION_INPUTS_32BIT.TcDUT

TYPE MNG_APPLICATION_INPUTS_32BIT :
STRUCT
    NumSignals                     : INT     := 12        ;
    Cocktail_Holder1_00_VACUUM : BOOL    := 0; (* r_Adapter/Cocktail_Holder_1/Cocktail_Holder1?Vacuum *)
    DetectionCookieAdapter1_00_IR : BOOL    := 0; (* dapter/Cocktail_Holder_1/DetectionCookieAdapter1?IR *)
    Cocktail_Holder2_00_VACUUM : BOOL    := 0; (* r_Adapter/Cocktail_Holder_2/Cocktail_Holder2?Vacuum *)
    DetectionCookieAdapter2_00_IR : BOOL    := 0; (* dapter/Cocktail_Holder_2/DetectionCookieAdapter2?IR *)
    Cocktail_Holder3_00_VACUUM : BOOL    := 0; (* r_Adapter/Cocktail_Holder_3/Cocktail_Holder3?Vacuum *)
    DetectionCookieAdapter3_00_IR : BOOL    := 0; (* dapter/Cocktail_Holder_3/DetectionCookieAdapter3?IR *)
    Cocktail_Holder4_00_VACUUM : BOOL    := 0; (* r_Adapter/Cocktail_Holder_4/Cocktail_Holder4?Vacuum *)
    DetectionCookieAdapter4_00_IR : BOOL    := 0; (* dapter/Cocktail_Holder_4/DetectionCookieAdapter4?IR *)
    Cocktail_Holder5_00_VACUUM : BOOL    := 0; (* r_Adapter/Cocktail_Holder_5/Cocktail_Holder5?Vacuum *)
    DetectionCookieAdapter5_00_IR : BOOL    := 0; (* dapter/Cocktail_Holder_5/DetectionCookieAdapter5?IR *)
    Cocktail_Holder6_00_VACUUM : BOOL    := 0; (* r_Adapter/Cocktail_Holder_6/Cocktail_Holder6?Vacuum *)
    DetectionCookieAdapter6_00_IR : BOOL    := 0; (* dapter/Cocktail_Holder_6/DetectionCookieAdapter6?IR *)
END_STRUCT
END_TYPE

// ---- DUTs/industrialPhysics/MNG_APPLICATION_OUTPUTS_32BIT.TcDUT

TYPE MNG_APPLICATION_OUTPUTS_32BIT :
STRUCT
    NumSignals                     : INT     := 222       ;
    Fahrachse1_00_ChainDrvActual : REAL    := 0.0; (* Physics://physics/Fahrachse1?ChainDrvActual *)
    Cocktail_Holder_1_00_ACT_POS : REAL    := 0.0; (* /physics1/Mover_Adapter/Cocktail_Holder_1?KinActual *)
    Cocktail_Holder1_00_Priority : UDINT   := 0; (* Adapter/Cocktail_Holder_1/Cocktail_Holder1?Priority *)
    Cocktail_Holder1_00_GRIP : BOOL    := 0; (* _Adapter/Cocktail_Holder_1/Cocktail_Holder1?Gripper *)
    Fahrachse2_00_ChainDrvActual : REAL    := 0.0; (* Physics://physics/Fahrachse2?ChainDrvActual *)
    Cocktail_Holder_2_00_ACT_POS : REAL    := 0.0; (* /physics2/Mover_Adapter/Cocktail_Holder_2?KinActual *)
    Cocktail_Holder2_00_Priority : UDINT   := 0; (* Adapter/Cocktail_Holder_2/Cocktail_Holder2?Priority *)
    Cocktail_Holder2_00_GRIP : BOOL    := 0; (* _Adapter/Cocktail_Holder_2/Cocktail_Holder2?Gripper *)
    Fahrachse3_00_ChainDrvActual : REAL    := 0.0; (* Physics://physics/Fahrachse3?ChainDrvActual *)
    Cocktail_Holder_3_00_ACT_POS : REAL    := 0.0; (* /physics3/Mover_Adapter/Cocktail_Holder_3?KinActual *)
    Cocktail_Holder3_00_Priority : UDINT   := 0; (* Adapter/Cocktail_Holder_3/Cocktail_Holder3?Priority *)
    Cocktail_Holder3_00_GRIP : BOOL    := 0; (* _Adapter/Cocktail_Holder_3/Cocktail_Holder3?Gripper *)
    Fahrachse4_00_ChainDrvActual : REAL    := 0.0; (* Physics://physics/Fahrachse4?ChainDrvActual *)
    Cocktail_Holder_4_00_ACT_POS : REAL    := 0.0; (* /physics4/Mover_Adapter/Cocktail_Holder_4?KinActual *)
    Cocktail_Holder4_00_Priority : UDINT   := 0; (* Adapter/Cocktail_Holder_4/Cocktail_Holder4?Priority *)
    Cocktail_Holder4_00_GRIP : BOOL    := 0; (* _Adapter/Cocktail_Holder_4/Cocktail_Holder4?Gripper *)
    Fahrachse5_00_ChainDrvActual : REAL    := 0.0; (* Physics://physics/Fahrachse5?ChainDrvActual *)
    Cocktail_Holder_5_00_ACT_POS : REAL    := 0.0; (* /physics5/Mover_Adapter/Cocktail_Holder_5?KinActual *)
    Cocktail_Holder5_00_Priority : UDINT   := 0; (* Adapter/Cocktail_Holder_5/Cocktail_Holder5?Priority *)
    Cocktail_Holder5_00_GRIP : BOOL    := 0; (* _Adapter/Cocktail_Holder_5/Cocktail_Holder5?Gripper *)
    Fahrachse6_00_ChainDrvActual : REAL    := 0.0; (* Physics://physics/Fahrachse6?ChainDrvActual *)
    Cocktail_Holder_6_00_ACT_POS : REAL    := 0.0; (* /physics6/Mover_Adapter/Cocktail_Holder_6?KinActual *)
    Cocktail_Holder6_00_Priority : UDINT   := 0; (* Adapter/Cocktail_Holder_6/Cocktail_Holder6?Priority *)
    Cocktail_Holder6_00_GRIP : BOOL    := 0; (* _Adapter/Cocktail_Holder_6/Cocktail_Holder6?Gripper *)
    LED_2_65_00_on1 : BOOL    := 0; (* Physics://physics/LED2-3.5/LED_2.65?on1 *)
    LED_2_65_00_on2 : BOOL    := 0; (* Physics://physics/LED2-3.5/LED_2.65?on2 *)
    LED_2_65_00_on3 : BOOL    := 0; (* Physics://physics/LED2-3.5/LED_2.65?on3 *)
    LED_2_60_00_on1 : BOOL    := 0; (* Physics://physics/LED2-3.5/LED_2.60?on1 *)
    LED_2_60_00_on2 : BOOL    := 0; (* Physics://physics/LED2-3.5/LED_2.60?on2 *)
    LED_2_60_00_on3 : BOOL    := 0; (* Physics://physics/LED2-3.5/LED_2.60?on3 *)
    LED_3_05_00_on1 : BOOL    := 0; (* Physics://physics/LED2-3.5/LED_3.05?on1 *)
    LED_3_05_00_on2 : BOOL    := 0; (* Physics://physics/LED2-3.5/LED_3.05?on2 *)
    LED_3_05_00_on3 : BOOL    := 0; (* Physics://physics/LED2-3.5/LED_3.05?on3 *)
    LED_2_50_00_on1 : BOOL    := 0; (* Physics://physics/LED2-3.5/LED_2.50?on1 *)
    LED_2_50_00_on2 : BOOL    := 0; (* Physics://physics/LED2-3.5/LED_2.50?on2 *)
    LED_2_50_00_on3 : BOOL    := 0; (* Physics://physics/LED2-3.5/LED_2.50?on3 *)
    LED_2_55_00_on1 : BOOL    := 0; (* Physics://physics/LED2-3.5/LED_2.55?on1 *)
    LED_2_55_00_on2 : BOOL    := 0; (* Physics://physics/LED2-3.5/LED_2.55?on2 *)
    LED_2_55_00_on3 : BOOL    := 0; (* Physics://physics/LED2-3.5/LED_2.55?on3 *)
    LED_3_00_00_on1 : BOOL    := 0; (* Physics://physics/LED2-3.5/LED_3.00?on1 *)
    LED_3_00_00_on2 : BOOL    := 0; (* Physics://physics/LED2-3.5/LED_3.00?on2 *)
    LED_3_00_00_on3 : BOOL    := 0; (* Physics://physics/LED2-3.5/LED_3.00?on3 *)
    LED_2_95_00_on1 : BOOL    := 0; (* Physics://physics/LED2-3.5/LED_2.95?on1 *)
    LED_2_95_00_on2 : BOOL    := 0; (* Physics://physics/LED2-3.5/LED_2.95?on2 *)
    LED_2_95_00_on3 : BOOL    := 0; (* Physics://physics/LED2-3.5/LED_2.95?on3 *)
    LED_2_90_00_on1 : BOOL    := 0; (* Physics://physics/LED2-3.5/LED_2.90?on1 *)
    LED_2_90_00_on2 : BOOL    := 0; (* Physics://physics/LED2-3.5/LED_2.90?on2 *)
    LED_2_90_00_on3 : BOOL    := 0; (* Physics://physics/LED2-3.5/LED_2.90?on3 *)
    LED_2_85_00_on1 : BOOL    := 0; (* Physics://physics/LED2-3.5/LED_2.85?on1 *)
    LED_2_85_00_on2 : BOOL    := 0; (* Physics://physics/LED2-3.5/LED_2.85?on2 *)
    LED_2_85_00_on3 : BOOL    := 0; (* Physics://physics/LED2-3.5/LED_2.85?on3 *)
    LED_2_80_00_on1 : BOOL    := 0; (* Physics://physics/LED2-3.5/LED_2.80?on1 *)
    LED_2_80_00_on2 : BOOL    := 0; (* Physics://physics/LED2-3.5/LED_2.80?on2 *)
    LED_2_80_00_on3 : BOOL    := 0; (* Physics://physics/LED2-3.5/LED_2.80?on3 *)
    LED_2_75_00_on1 : BOOL    := 0; (* Physics://physics/LED2-3.5/LED_2.75?on1 *)
    LED_2_75_00_on2 : BOOL    := 0; (* Physics://physics/LED2-3.5/LED_2.75?on2 *)
    LED_2_75_00_on3 : BOOL    := 0; (* Physics://physics/LED2-3.5/LED_2.75?on3 *)
    LED_2_70_00_on1 : BOOL    := 0; (* Physics://physics/LED2-3.5/LED_2.70?on1 *)
    LED_2_70_00_on2 : BOOL    := 0; (* Physics://physics/LED2-3.5/LED_2.70?on2 *)
    LED_2_70_00_on3 : BOOL    := 0; (* Physics://physics/LED2-3.5/LED_2.70?on3 *)
    LED_3_10_00_on1 : BOOL    := 0; (* Physics://physics/LED2-3.5/LED_3.10?on1 *)
    LED_3_10_00_on2 : BOOL    := 0; (* Physics://physics/LED2-3.5/LED_3.10?on2 *)
    LED_3_10_00_on3 : BOOL    := 0; (* Physics://physics/LED2-3.5/LED_3.10?on3 *)
    LED_3_15_00_on1 : BOOL    := 0; (* Physics://physics/LED2-3.5/LED_3.15?on1 *)
    LED_3_15_00_on2 : BOOL    := 0; (* Physics://physics/LED2-3.5/LED_3.15?on2 *)
    LED_3_15_00_on3 : BOOL    := 0; (* Physics://physics/LED2-3.5/LED_3.15?on3 *)
    LED_3_20_00_on1 : BOOL    := 0; (* Physics://physics/LED2-3.5/LED_3.20?on1 *)
    LED_3_20_00_on2 : BOOL    := 0; (* Physics://physics/LED2-3.5/LED_3.20?on2 *)
    LED_3_20_00_on3 : BOOL    := 0; (* Physics://physics/LED2-3.5/LED_3.20?on3 *)
    LED_3_25_00_on1 : BOOL    := 0; (* Physics://physics/LED2-3.5/LED_3.25?on1 *)
    LED_3_25_00_on2 : BOOL    := 0; (* Physics://physics/LED2-3.5/LED_3.25?on2 *)
    LED_3_25_00_on3 : BOOL    := 0; (* Physics://physics/LED2-3.5/LED_3.25?on3 *)
    LED_3_45_00_on1 : BOOL    := 0; (* Physics://physics/LED2-3.5/LED_3.45?on1 *)
    LED_3_45_00_on2 : BOOL    := 0; (* Physics://physics/LED2-3.5/LED_3.45?on2 *)
    LED_3_45_00_on3 : BOOL    := 0; (* Physics://physics/LED2-3.5/LED_3.45?on3 *)
    LED_3_40_00_on1 : BOOL    := 0; (* Physics://physics/LED2-3.5/LED_3.40?on1 *)
    LED_3_40_00_on2 : BOOL    := 0; (* Physics://physics/LED2-3.5/LED_3.40?on2 *)
    LED_3_40_00_on3 : BOOL    := 0; (* Physics://physics/LED2-3.5/LED_3.40?on3 *)
    LED_2_25_00_on1 : BOOL    := 0; (* Physics://physics/LED2-3.5/LED_2.25?on1 *)
    LED_2_25_00_on2 : BOOL    := 0; (* Physics://physics/LED2-3.5/LED_2.25?on2 *)
    LED_2_25_00_on3 : BOOL    := 0; (* Physics://physics/LED2-3.5/LED_2.25?on3 *)
    LED_2_20_00_on1 : BOOL    := 0; (* Physics://physics/LED2-3.5/LED_2.20?on1 *)
    LED_2_20_00_on2 : BOOL    := 0; (* Physics://physics/LED2-3.5/LED_2.20?on2 *)
    LED_2_20_00_on3 : BOOL    := 0; (* Physics://physics/LED2-3.5/LED_2.20?on3 *)
    LED_2_15_00_on1 : BOOL    := 0; (* Physics://physics/LED2-3.5/LED_2.15?on1 *)
    LED_2_15_00_on2 : BOOL    := 0; (* Physics://physics/LED2-3.5/LED_2.15?on2 *)
    LED_2_15_00_on3 : BOOL    := 0; (* Physics://physics/LED2-3.5/LED_2.15?on3 *)
    LED_2_10_00_on1 : BOOL    := 0; (* Physics://physics/LED2-3.5/LED_2.10?on1 *)
    LED_2_10_00_on2 : BOOL    := 0; (* Physics://physics/LED2-3.5/LED_2.10?on2 *)
    LED_2_10_00_on3 : BOOL    := 0; (* Physics://physics/LED2-3.5/LED_2.10?on3 *)
    LED_2_05_00_on1 : BOOL    := 0; (* Physics://physics/LED2-3.5/LED_2.05?on1 *)
    LED_2_05_00_on2 : BOOL    := 0; (* Physics://physics/LED2-3.5/LED_2.05?on2 *)
    LED_2_05_00_on3 : BOOL    := 0; (* Physics://physics/LED2-3.5/LED_2.05?on3 *)
    LED_2_00_00_on1 : BOOL    := 0; (* Physics://physics/LED2-3.5/LED_2.00?on1 *)
    LED_2_00_00_on2 : BOOL    := 0; (* Physics://physics/LED2-3.5/LED_2.00?on2 *)
    LED_2_00_00_on3 : BOOL    := 0; (* Physics://physics/LED2-3.5/LED_2.00?on3 *)
    LED_3_35_00_on1 : BOOL    := 0; (* Physics://physics/LED2-3.5/LED_3.35?on1 *)
    LED_3_35_00_on2 : BOOL    := 0; (* Physics://physics/LED2-3.5/LED_3.35?on2 *)
    LED_3_35_00_on3 : BOOL    := 0; (* Physics://physics/LED2-3.5/LED_3.35?on3 *)
    LED_3_30_00_on1 : BOOL    := 0; (* Physics://physics/LED2-3.5/LED_3.30?on1 *)
    LED_3_30_00_on2 : BOOL    := 0; (* Physics://physics/LED2-3.5/LED_3.30?on2 *)
    LED_3_30_00_on3 : BOOL    := 0; (* Physics://physics/LED2-3.5/LED_3.30?on3 *)
    LED_2_35_00_on1 : BOOL    := 0; (* Physics://physics/LED2-3.5/LED_2.35?on1 *)
    LED_2_35_00_on2 : BOOL    := 0; (* Physics://physics/LED2-3.5/LED_2.35?on2 *)
    LED_2_35_00_on3 : BOOL    := 0; (* Physics://physics/LED2-3.5/LED_2.35?on3 *)
    LED_2_30_00_on1 : BOOL    := 0; (* Physics://physics/LED2-3.5/LED_2.30?on1 *)
    LED_2_30_00_on2 : BOOL    := 0; (* Physics://physics/LED2-3.5/LED_2.30?on2 *)
    LED_2_30_00_on3 : BOOL    := 0; (* Physics://physics/LED2-3.5/LED_2.30?on3 *)
    LED_2_40_00_on1 : BOOL    := 0; (* Physics://physics/LED2-3.5/LED_2.40?on1 *)
    LED_2_40_00_on2 : BOOL    := 0; (* Physics://physics/LED2-3.5/LED_2.40?on2 *)
    LED_2_40_00_on3 : BOOL    := 0; (* Physics://physics/LED2-3.5/LED_2.40?on3 *)
    LED_2_45_00_on1 : BOOL    := 0; (* Physics://physics/LED2-3.5/LED_2.45?on1 *)
    LED_2_45_00_on2 : BOOL    := 0; (* Physics://physics/LED2-3.5/LED_2.45?on2 *)
    LED_2_45_00_on3 : BOOL    := 0; (* Physics://physics/LED2-3.5/LED_2.45?on3 *)
    LED_0_80_00_on1 : BOOL    := 0; (* Physics://physics/LED0-1.5/LED_0.80?on1 *)
    LED_0_80_00_on2 : BOOL    := 0; (* Physics://physics/LED0-1.5/LED_0.80?on2 *)
    LED_0_80_00_on3 : BOOL    := 0; (* Physics://physics/LED0-1.5/LED_0.80?on3 *)
    LED_0_85_00_on1 : BOOL    := 0; (* Physics://physics/LED0-1.5/LED_0.85?on1 *)
    LED_0_85_00_on2 : BOOL    := 0; (* Physics://physics/LED0-1.5/LED_0.85?on2 *)
    LED_0_85_00_on3 : BOOL    := 0; (* Physics://physics/LED0-1.5/LED_0.85?on3 *)
    LED_0_40_00_on1 : BOOL    := 0; (* Physics://physics/LED0-1.5/LED_0.40?on1 *)
    LED_0_40_00_on2 : BOOL    := 0; (* Physics://physics/LED0-1.5/LED_0.40?on2 *)
    LED_0_40_00_on3 : BOOL    := 0; (* Physics://physics/LED0-1.5/LED_0.40?on3 *)
    LED_0_95_00_on1 : BOOL    := 0; (* Physics://physics/LED0-1.5/LED_0.95?on1 *)
    LED_0_95_00_on2 : BOOL    := 0; (* Physics://physics/LED0-1.5/LED_0.95?on2 *)
    LED_0_95_00_on3 : BOOL    := 0; (* Physics://physics/LED0-1.5/LED_0.95?on3 *)
    LED_0_90_00_on1 : BOOL    := 0; (* Physics://physics/LED0-1.5/LED_0.90?on1 *)
    LED_0_90_00_on2 : BOOL    := 0; (* Physics://physics/LED0-1.5/LED_0.90?on2 *)
    LED_0_90_00_on3 : BOOL    := 0; (* Physics://physics/LED0-1.5/LED_0.90?on3 *)
    LED_0_45_00_on1 : BOOL    := 0; (* Physics://physics/LED0-1.5/LED_0.45?on1 *)
    LED_0_45_00_on2 : BOOL    := 0; (* Physics://physics/LED0-1.5/LED_0.45?on2 *)
    LED_0_45_00_on3 : BOOL    := 0; (* Physics://physics/LED0-1.5/LED_0.45?on3 *)
    LED_0_50_00_on1 : BOOL    := 0; (* Physics://physics/LED0-1.5/LED_0.50?on1 *)
    LED_0_50_00_on2 : BOOL    := 0; (* Physics://physics/LED0-1.5/LED_0.50?on2 *)
    LED_0_50_00_on3 : BOOL    := 0; (* Physics://physics/LED0-1.5/LED_0.50?on3 *)
    LED_0_55_00_on1 : BOOL    := 0; (* Physics://physics/LED0-1.5/LED_0.55?on1 *)
    LED_0_55_00_on2 : BOOL    := 0; (* Physics://physics/LED0-1.5/LED_0.55?on2 *)
    LED_0_55_00_on3 : BOOL    := 0; (* Physics://physics/LED0-1.5/LED_0.55?on3 *)
    LED_0_60_00_on1 : BOOL    := 0; (* Physics://physics/LED0-1.5/LED_0.60?on1 *)
    LED_0_60_00_on2 : BOOL    := 0; (* Physics://physics/LED0-1.5/LED_0.60?on2 *)
    LED_0_60_00_on3 : BOOL    := 0; (* Physics://physics/LED0-1.5/LED_0.60?on3 *)
    LED_0_65_00_on1 : BOOL    := 0; (* Physics://physics/LED0-1.5/LED_0.65?on1 *)
    LED_0_65_00_on2 : BOOL    := 0; (* Physics://physics/LED0-1.5/LED_0.65?on2 *)
    LED_0_65_00_on3 : BOOL    := 0; (* Physics://physics/LED0-1.5/LED_0.65?on3 *)
    LED_0_70_00_on1 : BOOL    := 0; (* Physics://physics/LED0-1.5/LED_0.70?on1 *)
    LED_0_70_00_on2 : BOOL    := 0; (* Physics://physics/LED0-1.5/LED_0.70?on2 *)
    LED_0_70_00_on3 : BOOL    := 0; (* Physics://physics/LED0-1.5/LED_0.70?on3 *)
    LED_0_75_00_on1 : BOOL    := 0; (* Physics://physics/LED0-1.5/LED_0.75?on1 *)
    LED_0_75_00_on2 : BOOL    := 0; (* Physics://physics/LED0-1.5/LED_0.75?on2 *)
    LED_0_75_00_on3 : BOOL    := 0; (* Physics://physics/LED0-1.5/LED_0.75?on3 *)
    LED_0_35_00_on1 : BOOL    := 0; (* Physics://physics/LED0-1.5/LED_0.35?on1 *)
    LED_0_35_00_on2 : BOOL    := 0; (* Physics://physics/LED0-1.5/LED_0.35?on2 *)
    LED_0_35_00_on3 : BOOL    := 0; (* Physics://physics/LED0-1.5/LED_0.35?on3 *)
    LED_0_30_00_on1 : BOOL    := 0; (* Physics://physics/LED0-1.5/LED_0.30?on1 *)
    LED_0_30_00_on2 : BOOL    := 0; (* Physics://physics/LED0-1.5/LED_0.30?on2 *)
    LED_0_30_00_on3 : BOOL    := 0; (* Physics://physics/LED0-1.5/LED_0.30?on3 *)
    LED_0_25_00_on1 : BOOL    := 0; (* Physics://physics/LED0-1.5/LED_0.25?on1 *)
    LED_0_25_00_on2 : BOOL    := 0; (* Physics://physics/LED0-1.5/LED_0.25?on2 *)
    LED_0_25_00_on3 : BOOL    := 0; (* Physics://physics/LED0-1.5/LED_0.25?on3 *)
    LED_0_20_00_on1 : BOOL    := 0; (* Physics://physics/LED0-1.5/LED_0.20?on1 *)
    LED_0_20_00_on2 : BOOL    := 0; (* Physics://physics/LED0-1.5/LED_0.20?on2 *)
    LED_0_20_00_on3 : BOOL    := 0; (* Physics://physics/LED0-1.5/LED_0.20?on3 *)
    LED_0_00_00_on1 : BOOL    := 0; (* Physics://physics/LED0-1.5/LED_0.00?on1 *)
    LED_0_00_00_on2 : BOOL    := 0; (* Physics://physics/LED0-1.5/LED_0.00?on2 *)
    LED_0_00_00_on3 : BOOL    := 0; (* Physics://physics/LED0-1.5/LED_0.00?on3 *)
    LED_0_05_00_on1 : BOOL    := 0; (* Physics://physics/LED0-1.5/LED_0.05?on1 *)
    LED_0_05_00_on2 : BOOL    := 0; (* Physics://physics/LED0-1.5/LED_0.05?on2 *)
    LED_0_05_00_on3 : BOOL    := 0; (* Physics://physics/LED0-1.5/LED_0.05?on3 *)
    LED_1_20_00_on1 : BOOL    := 0; (* Physics://physics/LED0-1.5/LED_1.20?on1 *)
    LED_1_20_00_on2 : BOOL    := 0; (* Physics://physics/LED0-1.5/LED_1.20?on2 *)
    LED_1_20_00_on3 : BOOL    := 0; (* Physics://physics/LED0-1.5/LED_1.20?on3 *)
    LED_1_25_00_on1 : BOOL    := 0; (* Physics://physics/LED0-1.5/LED_1.25?on1 *)
    LED_1_25_00_on2 : BOOL    := 0; (* Physics://physics/LED0-1.5/LED_1.25?on2 *)
    LED_1_25_00_on3 : BOOL    := 0; (* Physics://physics/LED0-1.5/LED_1.25?on3 *)
    LED_1_30_00_on1 : BOOL    := 0; (* Physics://physics/LED0-1.5/LED_1.30?on1 *)
    LED_1_30_00_on2 : BOOL    := 0; (* Physics://physics/LED0-1.5/LED_1.30?on2 *)
    LED_1_30_00_on3 : BOOL    := 0; (* Physics://physics/LED0-1.5/LED_1.30?on3 *)
    LED_1_35_00_on1 : BOOL    := 0; (* Physics://physics/LED0-1.5/LED_1.35?on1 *)
    LED_1_35_00_on2 : BOOL    := 0; (* Physics://physics/LED0-1.5/LED_1.35?on2 *)
    LED_1_35_00_on3 : BOOL    := 0; (* Physics://physics/LED0-1.5/LED_1.35?on3 *)
    LED_1_40_00_on1 : BOOL    := 0; (* Physics://physics/LED0-1.5/LED_1.40?on1 *)
    LED_1_40_00_on2 : BOOL    := 0; (* Physics://physics/LED0-1.5/LED_1.40?on2 *)
    LED_1_40_00_on3 : BOOL    := 0; (* Physics://physics/LED0-1.5/LED_1.40?on3 *)
    LED_1_45_00_on1 : BOOL    := 0; (* Physics://physics/LED0-1.5/LED_1.45?on1 *)
    LED_1_45_00_on2 : BOOL    := 0; (* Physics://physics/LED0-1.5/LED_1.45?on2 *)
    LED_1_45_00_on3 : BOOL    := 0; (* Physics://physics/LED0-1.5/LED_1.45?on3 *)
    LED_0_10_00_on1 : BOOL    := 0; (* Physics://physics/LED0-1.5/LED_0.10?on1 *)
    LED_0_10_00_on2 : BOOL    := 0; (* Physics://physics/LED0-1.5/LED_0.10?on2 *)
    LED_0_10_00_on3 : BOOL    := 0; (* Physics://physics/LED0-1.5/LED_0.10?on3 *)
    LED_0_15_00_on1 : BOOL    := 0; (* Physics://physics/LED0-1.5/LED_0.15?on1 *)
    LED_0_15_00_on2 : BOOL    := 0; (* Physics://physics/LED0-1.5/LED_0.15?on2 *)
    LED_0_15_00_on3 : BOOL    := 0; (* Physics://physics/LED0-1.5/LED_0.15?on3 *)
    LED_1_10_00_on1 : BOOL    := 0; (* Physics://physics/LED0-1.5/LED_1.10?on1 *)
    LED_1_10_00_on2 : BOOL    := 0; (* Physics://physics/LED0-1.5/LED_1.10?on2 *)
    LED_1_10_00_on3 : BOOL    := 0; (* Physics://physics/LED0-1.5/LED_1.10?on3 *)
    LED_1_15_00_on1 : BOOL    := 0; (* Physics://physics/LED0-1.5/LED_1.15?on1 *)
    LED_1_15_00_on2 : BOOL    := 0; (* Physics://physics/LED0-1.5/LED_1.15?on2 *)
    LED_1_15_00_on3 : BOOL    := 0; (* Physics://physics/LED0-1.5/LED_1.15?on3 *)
    LED_1_05_00_on1 : BOOL    := 0; (* Physics://physics/LED0-1.5/LED_1.05?on1 *)
    LED_1_05_00_on2 : BOOL    := 0; (* Physics://physics/LED0-1.5/LED_1.05?on2 *)
    LED_1_05_00_on3 : BOOL    := 0; (* Physics://physics/LED0-1.5/LED_1.05?on3 *)
    LED_1_00_00_on1 : BOOL    := 0; (* Physics://physics/LED0-1.5/LED_1.00?on1 *)
    LED_1_00_00_on2 : BOOL    := 0; (* Physics://physics/LED0-1.5/LED_1.00?on2 *)
    LED_1_00_00_on3 : BOOL    := 0; (* Physics://physics/LED0-1.5/LED_1.00?on3 *)
    Seitenwand_00_reserved_colour02 : BOOL    := 0; (* c/physics2/Mover_Adapter/Seitenwand?reserved_colour *)
    Seitenwand_00_blocked_colour02 : BOOL    := 0; (* ic/physics2/Mover_Adapter/Seitenwand?blocked_colour *)
    Seitenwand_00_error_colour02 : BOOL    := 0; (* blic/physics2/Mover_Adapter/Seitenwand?error_colour *)
    Seitenwand0_00_reserved_colour02 : BOOL    := 0; (* /physics2/Mover_Adapter/Seitenwand0?reserved_colour *)
    Seitenwand0_00_blocked_colour02 : BOOL    := 0; (* c/physics2/Mover_Adapter/Seitenwand0?blocked_colour *)
    Seitenwand0_00_error_colour02 : BOOL    := 0; (* lic/physics2/Mover_Adapter/Seitenwand0?error_colour *)
    Seitenwand_00_reserved_colour04 : BOOL    := 0; (* c/physics4/Mover_Adapter/Seitenwand?reserved_colour *)
    Seitenwand_00_blocked_colour04 : BOOL    := 0; (* ic/physics4/Mover_Adapter/Seitenwand?blocked_colour *)
    Seitenwand_00_error_colour04 : BOOL    := 0; (* blic/physics4/Mover_Adapter/Seitenwand?error_colour *)
    Seitenwand0_00_reserved_colour04 : BOOL    := 0; (* /physics4/Mover_Adapter/Seitenwand0?reserved_colour *)
    Seitenwand0_00_blocked_colour04 : BOOL    := 0; (* c/physics4/Mover_Adapter/Seitenwand0?blocked_colour *)
    Seitenwand0_00_error_colour04 : BOOL    := 0; (* lic/physics4/Mover_Adapter/Seitenwand0?error_colour *)
    Seitenwand_00_reserved_colour06 : BOOL    := 0; (* c/physics6/Mover_Adapter/Seitenwand?reserved_colour *)
    Seitenwand_00_blocked_colour06 : BOOL    := 0; (* ic/physics6/Mover_Adapter/Seitenwand?blocked_colour *)
    Seitenwand_00_error_colour06 : BOOL    := 0; (* blic/physics6/Mover_Adapter/Seitenwand?error_colour *)
    Seitenwand0_00_reserved_colour06 : BOOL    := 0; (* /physics6/Mover_Adapter/Seitenwand0?reserved_colour *)
    Seitenwand0_00_blocked_colour06 : BOOL    := 0; (* c/physics6/Mover_Adapter/Seitenwand0?blocked_colour *)
    Seitenwand0_00_error_colour06 : BOOL    := 0; (* lic/physics6/Mover_Adapter/Seitenwand0?error_colour *)
END_STRUCT
END_TYPE

// ---- DUTs/industrialPhysics/MNG_DataArray.TcDUT
TYPE MNG_DataArray :
ARRAY[1..MNG_BUFFER_SIZE] OF DWORD;
END_TYPE

// ---- DUTs/industrialPhysics/MNG_DatagramHeader.TcDUT
TYPE MNG_DatagramHeader :
STRUCT
	/// Time when datagram has been created 
	Counter: DWORD;
	/// Time when datagram has been sent 
	SentTime: DWORD;
	/// Type of the datagram 
	DatagramType: DWORD := MNG_UnknownDatagram;
	/// Byte count in the payload 
	ByteCount: DWORD := 0;
END_STRUCT
END_TYPE

// ---- DUTs/industrialPhysics/MNG_DatagramType.TcDUT
TYPE MNG_DatagramType :
(
	///Dead man datagram signalizing peer is alive 
	MNG_DeadManDatagram := 0,
	///Time tick synchonisation 
	MNG_TimeTick,
	///Time tick synchonisation 
	MNG_TimeTickRequest,
	///Initialization of the connection 
	MNG_InitConnection,
	///Reset simulation 
	MNG_ResetSimulation,
	///Rewind simulation 
	MNG_RewindSimulation,
	///Start simulation 
	MNG_StartSimulation,
	///Stop simulation 
	MNG_StopSimulation,
	///IO Config datagram 
	MNG_IOConfig,
	///Complete Raw IO Image 
	MNG_RawIOImage,
	///Complete Raw 32 Bit IO Image 
	MNG_Raw32BitImage,
	///Delta IO, only ios that have changed 
	/// IODelta, 
	///Text datagram 
	MNG_TextDatagram,
	///Unknown Datagram (future updates of peer, not supported by this side) 
	MNG_UnknownDatagram
);
END_TYPE

// ---- DUTs/industrialPhysics/MNG_POSE6.TcDUT
TYPE MNG_POSE6 :
STRUCT
	x: REAL;
	y: REAL;
	z: REAL;
	a: REAL;
	b: REAL;
	c: REAL;
END_STRUCT
END_TYPE

// ---- DUTs/industrialPhysics/MNG_RawDatagram.TcDUT
TYPE MNG_RawDatagram :
STRUCT
	/// datagram header 
	Header: MNG_DatagramHeader;
	Payload: MNG_DataARRAY;
END_STRUCT
END_TYPE

// ---- DUTs/industrialPhysics/VEC3.TcDUT
TYPE VEC3 :
STRUCT
	x: REAL;
	y: REAL;
	z: REAL;
END_STRUCT
END_TYPE

// ---- DUTs/In_outputmnoduklesimu/DUT_SimulationFeed.TcDUT
TYPE DUT_SimulationFeed :
STRUCT
	xPosition : ARRAY [0..10] OF LREAL;
	
END_STRUCT
END_TYPE

// ---- DUTs/OPC Data Structure/DUT_MODULE_INTERFACE.TcDUT
/// MODULE INTERFACE INPUT AND OUTPUT 
TYPE DUT_MODULE_INTERFACE :
STRUCT
	///Information that the module reads
	Input: DUT_MODULE_INTERFACE_INPUT;
	///Information that the module write
	Output: DUT_MODULE_INTERFACE_OUTPUT;
END_STRUCT
END_TYPE

// ---- DUTs/OPC Data Structure/DUT_MODULE_INTERFACE_INPUT.TcDUT
TYPE DUT_MODULE_INTERFACE_INPUT :
STRUCT
	///Mode to run (init,auto,manual,..)
	Mode: DUT_MODE;
	///check if the modules is alive
	ConnectionTestInput: BOOL;
	///Modules get their position
	PositionInput: LREAL;
	///Update data= TRUE, No updatedata=FALSE
	Watchbit: BOOL;
	///Emergency stop
	EmergencyStop: BOOL;
	///Range of INPUT skills
	SkillInput: ARRAY[0..SkillCnt] OF DUT_SKILL_INPUT;
END_STRUCT
END_TYPE

// ---- DUTs/OPC Data Structure/DUT_MODULE_INTERFACE_OUTPUT.TcDUT
TYPE DUT_MODULE_INTERFACE_OUTPUT :
STRUCT
	///Free to use = TRUE, busy to use =FALSE
	Dummy: BOOL := TRUE;
	///Individual name of the module
	Name: STRING(80);
	///Identification number of module
	ID: UINT;
	///IP address
	IP: STRING(80);
	///Show if the module is in Standby or not
	Idle: BOOL;
	///Show if the module is connected
	Connected: BOOL;
	///Feedback with conection test input
	ConnectionTestOutput: BOOL;
	///Show if the system has error when=TRUE
	Error: BOOL;
	///Identification number of the error
	ErrorID: UINT;
	///Description of the error
	ErrorDescription: STRING(80);
	///Description of the current task
	CurrentTaskDescription: STRING(80);
	///Position of the sensor
	PositionSensor: BOOL;
	///Range of OUTPUT skills
	SkillOutput: ARRAY[0..SkillCnt] OF DUT_SKILL_OUTPUT;
	///Range of state values
	StateValue: ARRAY[0..StateCnt] OF DUT_STATEVALUES;
END_STRUCT
END_TYPE

// ---- DUTs/OPC Data Structure/DUT_PARAMETER.TcDUT
TYPE DUT_PARAMETER :
STRUCT
	///Free to use = TRUE, busy to use =FALSE
	Dummy: BOOL;
	///ID of the parameter
	ID: UINT;
	///Name of the parameter
	Name: STRING(80);
	///Unit of the parameter (mm,L,...)
	Unit: STRING(80);
	///Optional parameter
	Required: BOOL;
	///Default parameter to work
	Default: LREAL;
	///Minimum value of the parameter
	MinValue: LREAL;
	///Maximum value of the parameter
	MaxValue: LREAL;
END_STRUCT
END_TYPE

// ---- DUTs/OPC Data Structure/DUT_SKILL.TcDUT
///  Skill variables inside DUT_TASK
TYPE DUT_SKILL :
STRUCT
	///Name assigned for the process tool
	AssignedModuleName: STRING(80);
	///ID assigned for the process tool
	AssignedModuleID: UINT;
	///Position assigned for the process tool
	AssignedModulePosition: STRING(80);
	///Free to use = TRUE, busy to use =FALSE
	Dummy: BOOL;
	///Identification number of the skill
	ID: UINT;
	///Name of the skill
	Name: STRING(80);
	///Range of parameters
	Parameter: ARRAY[0..StateCnt] OF DUT_PARAMETER;
END_STRUCT
END_TYPE

// ---- DUTs/OPC Data Structure/DUT_SKILL_INPUT.TcDUT
TYPE DUT_SKILL_INPUT :
STRUCT
	///Range of parameters
	ParameterInput: ARRAY[0..ParameterCnt] OF DUT_PARAMETER_INPUT;
	///Start process
	Execute: BOOL;
END_STRUCT
END_TYPE

// ---- DUTs/OPC Data Structure/DUT_SKILL_OUTPUT.TcDUT
TYPE DUT_SKILL_OUTPUT :
STRUCT
	//Free to use = TRUE, busy to use =FALSE
	Dummy: BOOL := TRUE;
	//Identification number of skill
	ID: UINT;
	//indentfication name of skill
	Name: STRING(80);
	//Skill activated
	Activated: BOOL;
	//Ready to do skill
	Ready: BOOL;
	//Skill in process
	Busy: BOOL;
	//Skill finish
	Done: BOOL;
	//Error in system
	Error: BOOL;
	//Range of parameters
	ParameterOutput: ARRAY[0..ParameterCnt] OF DUT_PARAMETER_OUTPUT;
END_STRUCT
END_TYPE

// ---- DUTs/OPC Data Structure/DUT_TASK.TcDUT
TYPE DUT_TASK :
STRUCT
	///Name of the Task
	Name: STRING(80);
	///Free to use = TRUE, busy to use =FALSE
	Dummy: BOOL;
	///Identification number of the Task
	TaskID: INT;
	///Identification number of the Recipe
	RecipeID: INT;
	///Range of Skill in the TASK
	Skill: ARRAY[0..TaskSkillCnt] OF DUT_SKILL;
	///When occurs the action
	Timestamp: STRING(80);
	///State of the TASK e.g (unassigned, assigned, waitingForSkillReady, inProgress, done, aborted, error)
	State: DUT_TASKSTATE;
END_STRUCT
END_TYPE

// ---- DUTs/OPC Data Structure/DUT_TASKSTATE.TcDUT
TYPE DUT_TASKSTATE :
(
	Unassigned := 0,
	Assigned := 1,
	WaitingForSkillReady := 2,
	InProgress := 3,
	Done := 4,
	Aborted := 5,
	Error := 6
);
END_TYPE

// ---- DUTs/Server DUTs/Server DUTs/Server DUTs/DUT_MODE.TcDUT
/// MODE to run (inside of MODULE_INTERFACE_INPUT)
TYPE DUT_MODE :
(
	///Initialitzation number mode
	Init := 0,
	///Automatic number mode
	Auto := 1,
	///Manual number mode
	Manual := 2,
	Reset := 3
);
END_TYPE

// ---- DUTs/Server DUTs/Server DUTs/Server DUTs/DUT_PARAMETER_INPUT.TcDUT
TYPE DUT_PARAMETER_INPUT :
STRUCT
	///Value of the parameter 
	Value: LREAL;
	///Possibility to a string value depending on the parameter
	StringValue: STRING(80);
END_STRUCT
END_TYPE

// ---- DUTs/Server DUTs/Server DUTs/Server DUTs/DUT_PARAMETER_OUTPUT.TcDUT
TYPE DUT_PARAMETER_OUTPUT :
STRUCT
	///Free to use = TRUE, busy to use =FALSE
	Dummy: BOOL := TRUE;
	///ID of the parameter
	ID: UINT;
	///Name of the parameter
	Name: STRING(80);
	///Unit of the parameter
	Unit: STRING(80);
	///Optional parameter
	Required: BOOL;
	///Default parameter to work
	Default: LREAL;
	///Minimum value of the parameter
	MinValue: LREAL;
	///Maximum value of the parameter
	MaxValue: LREAL;
END_STRUCT
END_TYPE

// ---- DUTs/Server DUTs/Server DUTs/Server DUTs/DUT_SERVER_MODULE_INTERFACE.TcDUT
/// MODULE INTERFACE INPUT AND OUTPUT 
TYPE DUT_SERVER_MODULE_INTERFACE :
STRUCT
	///Information that the module reads
	Input: DUT_SERVER_MODULE_INTERFACE_INPUT;
	///Information that the module write
	Output: DUT_SERVER_MODULE_INTERFACE_OUTPUT;
END_STRUCT
END_TYPE

// ---- DUTs/Server DUTs/Server DUTs/Server DUTs/DUT_SERVER_MODULE_INTERFACE_INPUT.TcDUT
TYPE DUT_SERVER_MODULE_INTERFACE_INPUT :
STRUCT
	///Mode to run (init,auto,manual,..)
	Mode: INT;
	///check if the modules is alive
	ConnectionTestInput: BOOL;
	///Modules get their position
	PositionInput: LREAL;
	///Update data= TRUE, No updatedata=FALSE
	Watchbit: BOOL;
	///Emergency stop
	EmergencyStop: BOOL;
	///Range of INPUT skills
	SkillInput: DUT_SERVER_SKILLINPUTARRAY;
END_STRUCT
END_TYPE

// ---- DUTs/Server DUTs/Server DUTs/Server DUTs/DUT_SERVER_MODULE_INTERFACE_OUTPUT.TcDUT
TYPE DUT_SERVER_MODULE_INTERFACE_OUTPUT :
STRUCT
	///Free to use = TRUE, busy to use =FALSE
	Dummy: BOOL := TRUE;
	///Individual name of the module
	Name: STRING(80);
	///Identification number of module
	ID: UINT;
	///IP address
	IP: STRING(80);
	///Show if the module is in Standby or not
	Idle: BOOL;
	///Show if the module is connected
	Connected: BOOL;
	///Feedback with conection test input
	ConnectionTestOutput: BOOL;
	///Show if the system has error when=TRUE
	Error: BOOL;
	///Identification number of the error
	ErrorID: UINT;
	///Description of the error
	ErrorDescription: STRING(80);
	///Description of the current task
	CurrentTaskDescription: STRING(80);
	///Position of the output
	PositionOutput: LREAL;
	/// Bool value of the Sensor
	PositionSensor: BOOL;
	///Range of OUTPUT skills
	SkillOutput: DUT_SERVER_SKILLOUTPUTARRAY;
	///Range of state values
	StateValue: DUT_SERVER_STATEVALUEARRAY;
END_STRUCT
END_TYPE

// ---- DUTs/Server DUTs/Server DUTs/Server DUTs/DUT_SERVER_PARAMETERINPUTARRAY.TcDUT
TYPE DUT_SERVER_PARAMETERINPUTARRAY :
STRUCT
	ParameterInput0: DUT_PARAMETER_INPUT;
	ParameterInput1: DUT_PARAMETER_INPUT;
	ParameterInput2: DUT_PARAMETER_INPUT;
	ParameterInput3: DUT_PARAMETER_INPUT;
	ParameterInput4: DUT_PARAMETER_INPUT;
	ParameterInput5: DUT_PARAMETER_INPUT;
END_STRUCT
END_TYPE

// ---- DUTs/Server DUTs/Server DUTs/Server DUTs/DUT_SERVER_PARAMETEROUTPUTARRAY.TcDUT
TYPE DUT_SERVER_PARAMETEROUTPUTARRAY :
STRUCT
	ParameterOutput0: DUT_PARAMETER_OUTPUT;
	ParameterOutput1: DUT_PARAMETER_OUTPUT;
	ParameterOutput2: DUT_PARAMETER_OUTPUT;
	ParameterOutput3: DUT_PARAMETER_OUTPUT;
	ParameterOutput4: DUT_PARAMETER_OUTPUT;
	ParameterOutput5: DUT_PARAMETER_OUTPUT;
END_STRUCT
END_TYPE

// ---- DUTs/Server DUTs/Server DUTs/Server DUTs/DUT_SERVER_SKILLINPUTARRAY.TcDUT
TYPE DUT_SERVER_SKILLINPUTARRAY :
STRUCT
	SkillInput0: DUT_SERVER_SKILL_INPUT;
	SkillInput1: DUT_SERVER_SKILL_INPUT;
	SkillInput2: DUT_SERVER_SKILL_INPUT;
	SkillInput3: DUT_SERVER_SKILL_INPUT;
	SkillInput4: DUT_SERVER_SKILL_INPUT;
	SkillInput5: DUT_SERVER_SKILL_INPUT;
	SkillInput6: DUT_SERVER_SKILL_INPUT;
	SkillInput7: DUT_SERVER_SKILL_INPUT;
	SkillInput8: DUT_SERVER_SKILL_INPUT;
	SkillInput9: DUT_SERVER_SKILL_INPUT;
	SkillInput10: DUT_SERVER_SKILL_INPUT;
	SkillInput11: DUT_SERVER_SKILL_INPUT;
	SkillInput12: DUT_SERVER_SKILL_INPUT;
	SkillInput13: DUT_SERVER_SKILL_INPUT;
	SkillInput14: DUT_SERVER_SKILL_INPUT;
	SkillInput15: DUT_SERVER_SKILL_INPUT;
END_STRUCT
END_TYPE

// ---- DUTs/Server DUTs/Server DUTs/Server DUTs/DUT_SERVER_SKILLOUTPUTARRAY.TcDUT
TYPE DUT_SERVER_SKILLOUTPUTARRAY :
STRUCT
	SkillOutput0: DUT_SERVER_SKILL_OUTPUT;
	SkillOutput1: DUT_SERVER_SKILL_OUTPUT;
	SkillOutput2: DUT_SERVER_SKILL_OUTPUT;
	SkillOutput3: DUT_SERVER_SKILL_OUTPUT;
	SkillOutput4: DUT_SERVER_SKILL_OUTPUT;
	SkillOutput5: DUT_SERVER_SKILL_OUTPUT;
	SkillOutput6: DUT_SERVER_SKILL_OUTPUT;
	SkillOutput7: DUT_SERVER_SKILL_OUTPUT;
	SkillOutput8: DUT_SERVER_SKILL_OUTPUT;
	SkillOutput9: DUT_SERVER_SKILL_OUTPUT;
	SkillOutput10: DUT_SERVER_SKILL_OUTPUT;
	SkillOutput11: DUT_SERVER_SKILL_OUTPUT;
	SkillOutput12: DUT_SERVER_SKILL_OUTPUT;
	SkillOutput13: DUT_SERVER_SKILL_OUTPUT;
	SkillOutput14: DUT_SERVER_SKILL_OUTPUT;
	SkillOutput15: DUT_SERVER_SKILL_OUTPUT;
END_STRUCT
END_TYPE

// ---- DUTs/Server DUTs/Server DUTs/Server DUTs/DUT_SERVER_SKILL_INPUT.TcDUT
TYPE DUT_SERVER_SKILL_INPUT :
STRUCT
	///Range of parameters
	ParameterInput: DUT_SERVER_PARAMETERINPUTARRAY;
	///Start process
	Execute: BOOL;
END_STRUCT
END_TYPE

// ---- DUTs/Server DUTs/Server DUTs/Server DUTs/DUT_SERVER_SKILL_OUTPUT.TcDUT
TYPE DUT_SERVER_SKILL_OUTPUT :
STRUCT
	///Free to use = TRUE, busy to use =FALSE
	Dummy: BOOL := TRUE;
	///Identification number of skill
	ID: UINT;
	///indentfication name of skill
	Name: STRING(80);
	///Skill activated
	Activated: BOOL;
	///Ready to do skill
	Ready: BOOL;
	///Skill in process
	Busy: BOOL;
	///Skill finish
	Done: BOOL;
	///Error in system
	Error: BOOL;
	///Range of parameters
	ParameterOutput: DUT_SERVER_PARAMETEROUTPUTARRAY;
END_STRUCT
END_TYPE

// ---- DUTs/Server DUTs/Server DUTs/Server DUTs/DUT_SERVER_STATEVALUEARRAY.TcDUT
TYPE DUT_SERVER_STATEVALUEARRAY :
STRUCT
	StateValue0: DUT_STATEVALUES;
	StateValue1: DUT_STATEVALUES;
	StateValue2: DUT_STATEVALUES;
	StateValue3: DUT_STATEVALUES;
	StateValue4: DUT_STATEVALUES;
	StateValue5: DUT_STATEVALUES;
	StateValue6: DUT_STATEVALUES;
	StateValue7: DUT_STATEVALUES;
	StateValue8: DUT_STATEVALUES;
	StateValue9: DUT_STATEVALUES;
	StateValue10: DUT_STATEVALUES;
END_STRUCT
END_TYPE

// ---- DUTs/Server DUTs/Server DUTs/Server DUTs/DUT_STATEVALUES.TcDUT
TYPE DUT_STATEVALUES :
STRUCT
	///Free to use = TRUE, busy to use =FALSE
	Dummy: BOOL := TRUE;
	///Value of the State
	Value: LREAL;
	///Name of the state
	Name: STRING(80);
	///Description of the state
	Description: STRING(80);
	///Unit of the state ()
	Unit: STRING(80);
END_STRUCT
END_TYPE

// ---- DUTs/XTS DUTs/DUT_MoverInfo.TcDUT
TYPE DUT_MoverInfo :
STRUCT
	preposition: LREAL;
	postposition: LREAL;
	reserved: BOOL;
	blocked: BOOL;
	surpressed: BOOL;
	nocurvestop	: BOOL;
	
	SurpressedPosition: LREAL;
	SupressedClockwise: BOOL := FALSE;
	TaskID: INT;
END_STRUCT
END_TYPE

// ---- DUTs/XTS DUTs/DUT_XTS_Interface.TcDUT
TYPE DUT_XTS_Interface :
STRUCT
	Targetpos: LREAL;
	Setpos: LREAL;
	Buddygap	: LREAL;
	Buddyenable	: BOOL;
	Buddyactive	: BOOL;
	MovementDone: BOOL;
	Clockwise: BOOL;
	Velocity: LREAL;
	Acceleration: LREAL;
END_STRUCT
END_TYPE

// ---- GVLs/CAInterface.TcGVL
VAR_GLOBAL
	MoverInterface: ARRAY[1..grpcnt] OF DUT_XTS_Interface;
END_VAR

// ---- GVLs/GVL.TcGVL
VAR_GLOBAL
	ax: ARRAY[1..axcnt] OF AXIS_REF;
	poweredaxes	: ARRAY [1..axcnt] OF BOOL := [TRUE,TRUE,TRUE,TRUE,TRUE,TRUE];
	grp: ARRAY[1..grpcnt] OF AXIS_REF;
	CAgrp: CAGROUP_REF;
	/// OID of PollCallProxy, set via "Symbol Initialization" Tab in Instance of this PLC Project
	{attribute 'TcInitSymbol' := ''}
	callTargetOID : OTCID ;
	
	couplegap	: LREAL := 137;
	zerohightdistance	: LREAL := 132.82;
	CAgap		: LREAL	:= 200;
	
	
	buddyvelo	: LREAL		:= 30;
	freevelo	: LREAL		:= 500.0;
	maxvelo		: LREAL		:= 1500.0;
	defaultvelo	: LREAL		:= 500.0;
	freeacc		: LREAL		:= 8000.0;
	maxacc		: LREAL		:= 8000.0;
	defaulacc	: LREAL		:= 7800.0;
	initvelo	: LREAL		:= 300;
	nocurvesvelo	: LREAL := 350;
	surpressinggap	: LREAL := 200;
	
	restartstate	: INT := 0;
	
	bInput				: BOOL;
	//bSensor				: BOOL := 0; //OPC SENSOR INPUT
	measurementCycles	: INT := 4;
	MeasuredPosition	: ARRAY [1..10]OF LREAL;
	AveragedPosition	: LREAL := 13377.773;
	
	//OPC CLient GVL
	ClientSensorValue		: BOOL;
	ClientExecute			: BOOL;
	ClientReadEstablished	: BOOL;
	ClientDone				: BOOL;
	ClientWrite				: BOOL;
	ClientModuleServerUrl 	: STRING := 'opc.tcp://127.0.0.1:4840'; //'opc.tcp://192.168.175.224:4840';
	ClientReadIdentifier	: STRING := 'MI5.Module1102.Output.PositionSensor';
	ClientWriteIdentifier	: STRING:= 'MI5.Module1102.Input.PositionInput';
	ClientNamespaceIndex	: UINT;
	ClientNamespaceUri		: STRING;
	// Simulation Reserve Visu
	LampInterface			: ARRAY[1..ColourCnt] OF ARRAY [1..LampCnt] OF BOOL;
	
	
	CurveSection	: ARRAY [0..curvesectioncnt] OF LREAL := [1400,		1500, 	1562.5,		1625.0,		1687.5,		1750,		1812.5,		1875,		1937.5,		2000,		2100] ;
	CurveVelo		: ARRAY [0..curvesectioncnt] OF LREAL := [300,		300,	275,		250,		225,		200,		225,		250,		275,		300,		300] ;
	
	
END_VAR

VAR_GLOBAL CONSTANT
	raillength: LREAL := 4000.0;
	axcnt: UINT := 6;
	grpcnt: UINT := 3;
	curvesectioncnt	: UINT := 10;	
	// simu visu lampen:
	LampCnt					: UINT := 80;
	ColourCnt				: UINT := 4;
END_VAR

// ---- GVLs/industrialPhysics/MNG_GLOBALS.TcGVL
 VAR_GLOBAL CONSTANT
	/// Max. number of server<->client connections 
	PLCPRJ_MAX_CONNECTIONS: UDINT := 5;
	PLCPRJ_SERVER_RESPONSE_TIMEOUT: TIME := TIME#10s0ms;
	PLCPRJ_CLIENT_SEND_CYCLE_TIME: TIME := TIME#1ms;
	PLCPRJ_RECEIVER_POLLING_CYCLE_TIME: TIME := TIME#1ms;
	/// Max. internal fifo/receiver buffer size 
	PLCPRJ_BUFFER_SIZE: UDINT := 10000;
	/// receive fifo/buffer overflow
	PLCPRJ_ERROR_RECEIVE_BUFFER_OVERFLOW: UDINT := 16#8101;
	/// send fifo/buffer overflow 
	PLCPRJ_ERROR_SEND_BUFFER_OVERFLOW: UDINT := 16#8102;
	/// receive timeout error 
	PLCPRJ_ERROR_RESPONSE_TIMEOUT: UDINT := 16#8103;
	/// invalid frame format/data 
	PLCPRJ_ERROR_INVALID_FRAME_FORMAT: UDINT := 16#8104;
	/// invalid io format/data 
	PLCPRJ_ERROR_INVALID_IO_FORMAT_RECEIVED: UDINT := 16#8105;
	/// internal error 
	PLCPRJ_ERROR_INTERNAL: UDINT := 16#8105;
	/// rx data inconsistent 
	PLCPRJ_ERROR_RX_DATA_INCONSISTENT: UDINT := 16#8106;
	PLCPRJ_ERROR_RECEIVE_TIMEOUT: UDINT := 16#8107;
	/// send fifo overflow error 
	PLCPRJ_ERROR_SENDFIFO_OVERFLOW: UDINT := 16#8108;
	/// receive fifo overflow error 
	PLCPRJ_ERROR_RECFIFO_OVERFLOW: UDINT := 16#8109;
	/// Bytes: 131072; Max 128 KB of datagram payload data
	MNG_BUFFER_SIZE: DWORD := 32768;
	/// Max 10 datagrams buffered before loss occurs 
	MNG_DatagramsFIFO_Size: DWORD := 10;
	MNG_EmptyDatagramHeader: MNG_DatagramHeader;
	MNG_Application_NumInputs: DWORD := 4;
	MNG_Application_NumOutputs: DWORD := 4;
	/// PI should be defined by the system 
	/// PI      : LREAL := 3.1415926535897932384626433832795; 
	DEG2RAD: LREAL := 0.017453292519943295;
	RAD2DEG: LREAL := 57.295779513082323;
	MNG_TIMESTAMP: LREAL := 0;
END_VAR

// ---- GVLs/MI5.TcGVL
VAR_GLOBAL
	{attribute 'OPC.UA.DA' := '1'}
	Module2001: DUT_SERVER_MODULE_INTERFACE; 
	{attribute 'OPC.UA.DA' := '1'}
	Module2002: DUT_SERVER_MODULE_INTERFACE;
	{attribute 'OPC.UA.DA' := '1'}
	Module2003: DUT_SERVER_MODULE_INTERFACE;
	{attribute 'OPC.UA.DA' := '1'}
	ResetXTS	: BOOL;
	{attribute 'OPC.UA.DA' := '1'}
	Maintenance	: BOOL;
	{attribute 'OPC.UA.DA' := '1'}
	Restart		: BOOL;
	
	
END_VAR

// ---- GVLs/OPCConstants.TcGVL
VAR_GLOBAL CONSTANT
	///Maximum number of skillparameters
	ParameterCnt: INT := 5;
	///Maximum number of skills per Module
	SkillCnt: INT := 15;
	///Maximum number of Statevalues of one Module
	StateCnt: INT := 10;
	///Maximum number of modules
	
	
	
	ModuleCnt: INT := 10;
	///Maximum number of Tasks in Production List
	TaskCnt: INT := 30;
	///Maximum number  of offered recipes
	OfferCnt: INT := 5;
	///Maximum number of Orders in Queue
	OrderCnt: INT := 5;
	///Number of user set parameters per recipe
	UserParameterCnt: INT := 5;
	///Number of skills per task
	TaskSkillCnt: INT := 50;
END_VAR

// ---- GVLs/SKillGVL/ModuleInterface.TcGVL
VAR_GLOBAL
	Module		: ARRAY [1..GrpCnt] OF DUT_MODULE_INTERFACE;
	
END_VAR

// ---- GVLs/SKillGVL/Mover_Infos.TcGVL
VAR_GLOBAL
	MoverInfo: ARRAY[1..GrpCnt] OF DUT_MoverInfo;
	AwaitingReservationAxis: INT := 0;
	AwaitingAxisCnt: INT := 0;
	SkillAx:	ARRAY [1..GrpCnt] OF INT;
	Reservingaxis	: INT := 0;
	
END_VAR

// ---- GVLs/SKillGVL/SkillHandleConstants.TcGVL
VAR_GLOBAL
	WaySectionGap		: LREAL := 110.0;
	WaitingAbsPosition	: LREAL := 950;
	
	Startposition		: ARRAY[1..AxCnt] OF LREAL; // positionen, in denen sich die mover vor couple einfinden
END_VAR

// ---- POUs/OPC_Client.TcPOU
PROGRAM OPC_Client
VAR
	state 				: INT := 0;
	//fbOpen				: FB_OpcUAOpen;
	fbConnect			: FB_OPCServerConnect;
	fbReadVariable		: FB_ReadVariableOnce;
	fbWriteVariableOnce	: FB_WriteVariableOnce;
	
	// OPC INtern:
	ConnectionHandle	: DWORD;
	NamespaceIndex		: UINT;
	OPCTimer			: TON;
	OPCTimerout			: TIME;
END_VAR

IF ClientExecute THEN
	ClientDone := FALSE;
	NamespaceIndex := ClientNamespaceIndex;
	CASE state OF
		0:	state := 1;
			
		
		
		1:  
			fbConnect(ClientName := 'XTS',ServerUrl := ClientModuleServerUrl, NamespaceUri := ClientNamespaceUri,execute := TRUE, ConnectHdl => ConnectionHandle,Namespaceindex => NamespaceIndex);
			IF fbConnect.done THEN
			state := 2;
			END_IF
		2: 	fbReadVariable(ConnectionHdl := ConnectionHandle,IdentifierRead := ClientReadIdentifier,NamespaceIndex := ClientNamespaceIndex,execute := TRUE,SensorValue => ClientSensorValue);
			IF fbReadVariable.done THEN
				ClientReadEstablished := TRUE;
			END_IF
			IF ClientWrite THEN
				state := 5;
			END_IF
		
		
		5: 
			fbReadVariable(ConnectionHdl := ConnectionHandle,IdentifierRead := ClientReadIdentifier,NamespaceIndex := ClientNamespaceIndex,execute := TRUE,SensorValue => ClientSensorValue);
			fbWriteVariableOnce(
					IdentifierWrite:= ClientWriteIdentifier, 
					NamespaceIndex:= NamespaceIndex, 
					ConnectionHdl:= ConnectionHandle, 
					execute:= TRUE, 
					MeasuredPosition:= AveragedPosition, 
					done=> , 
					busy=> , 
					error=> );
			IF fbWriteVariableOnce.done THEN
				ClientDone := TRUE;
				ClientExecute := FALSE;
				state := 0;
			END_IF
	END_CASE
ELSE
fbConnect(execute := FALSE);
fbReadVariable(execute := FALSE);
fbWriteVariableOnce(execute := FALSE);
ClientReadEstablished := FALSE;
state := 0;
END_IF
bInput := ClientSensorValue;

END_PROGRAM

// ---- POUs/OPC Client/FB_OPCServerConnect.TcPOU
FUNCTION_BLOCK FB_OPCServerConnect
VAR_INPUT
	ServerUrl: STRING;
	NamespaceUri: STRING;
	ClientName: STRING;
	execute: BOOL;
END_VAR
VAR_OUTPUT
	ConnectHdl: DWORD;
	Namespaceindex: UINT;
	busy: BOOL;
	done: BOOL;
	error: BOOL;
END_VAR
VAR
	fbGetNameSpace: UA_GetNamespaceIndex;
	SesionconnectInfo: ST_UASessionConnectInfo;
	Timeout: TIME := DEFAULT_ADS_TIMEOUT;
	state: INT := -1;
	fbConnect: UA_Connect;
END_VAR

IF execute THEN
	CASE state OF
	-1: 	SesionconnectInfo.sApplicationName			:=ClientName;
			SesionconnectInfo.eSecurityMode				:=1; 
			SesionconnectInfo.eSecurityPolicyUri		:=1;
			SesionconnectInfo.eTransportProfileUri		:=1;
			SesionconnectInfo.tConnectTimeout			:=T#4S;
			SesionconnectInfo.tSessionTimeout			:=T#3S;
			
			
			busy 	:= TRUE;
			done	:= FALSE;							
			state 	:= 0;

	0:
         fbConnect(
			Execute:= FALSE, 
			ServerUrl:=ServerUrl , 
			SessionConnectInfo:= SesionconnectInfo, 
			Timeout:= Timeout, 
			ConnectionHdl=> ConnectHdl, 
			Done=>, 
			Busy=>busy, 
			Error=>error, 
			ErrorID=>);
			
	 		state := 1;
			
	1:
         fbConnect(
			Execute:= TRUE, 
			ServerUrl:=ServerUrl , 
			SessionConnectInfo:= SesionconnectInfo, 
			Timeout:= Timeout, 
			ConnectionHdl=> ConnectHdl,  
			Done=>, 
			Busy=>busy, 
			Error=>error, 
			ErrorID=> );
			
			IF fbConnect.done THEN
			
			state := 2;
			END_IF
		

			
 		
		
	2:	
		fbGetNameSpace(
			Execute:= FALSE,
			ConnectionHdl:=ConnectHdl,
			NamespaceUri:=NamespaceUri,
			Timeout:=Timeout,
			NamespaceIndex=>Namespaceindex,
			Done=>,
			Busy=>busy,
			Error=>error,
			ErrorID=>,);	
			
			state := 3;	
	3:
		fbGetNameSpace(
			Execute:= TRUE,
			ConnectionHdl:=ConnectHdl,
			NamespaceUri:=NamespaceUri,
			Timeout:=Timeout,
			NamespaceIndex=>Namespaceindex,
			Done=>,
			Busy=>busy,
			Error=>error,
			ErrorID=>,);
			IF fbGetNameSpace.done THEN
			Execute := FALSE;
			busy	:= FALSE;
			done	:= TRUE;
			state 	:= 0;
			END_IF
		END_CASE
ELSE 
state := -1;
END_IF

END_FUNCTION_BLOCK

// ---- POUs/OPC Client/FB_ReadVariableOnce.TcPOU
FUNCTION_BLOCK FB_ReadVariableOnce
VAR_INPUT
	IdentifierRead: STRING;
	NamespaceIndex: UINT;
	ConnectionHdl: DWORD;
	execute: BOOL;
END_VAR
VAR_OUTPUT
	SensorValue: BOOL;
	done: BOOL;
	busy: BOOL;
	error: BOOL;
END_VAR
VAR
	/// FBs
	fbNodeGetHandle: UA_NodeGetHandle;
	fbReadVariable: UA_Read;
	///Variables
	pSensorValue: POINTER TO BOOL;
	VariableSize: UDINT;
	NodeHdl: DWORD;
	cbDataR: UDINT;
	state: INT := -1;

	Timeout: TIME := DEFAULT_ADS_TIMEOUT;
	SessionNodeID	: ST_UANodeID;
END_VAR

IF execute THEN 
	CASE state OF
		
		-1:	SessionNodeID.nNamespaceIndex    			:= Namespaceindex;
			SessionNodeID.eIdentifierType				:= 1;
			SessionNodeID.sIdentifier					:= IdentifierRead;
			VariableSize 								:= SIZEOF (SensorValue);
			pSensorValue								:= ADR(SensorValue);
			
			
			

			busy := TRUE;
			done := FALSE;
			state:=0;

		0: fbNodeGetHandle(
			Execute:=FALSE,
			ConnectionHdl:=ConnectionHdl,
			NodeID:=SessionNodeID,
			Timeout:=Timeout,
			NodeHdl=>NodeHdl,
			Done=>,
			Busy=>busy,
			Error=>,
			ErrorID=>,);
			state:=1;
			
		1:fbNodeGetHandle(
			Execute:=TRUE,
			ConnectionHdl:=ConnectionHdl,
			NodeID:=SessionNodeID,
			Timeout:=Timeout,
			NodeHdl=>NodeHdl,
			Done=>,
			Busy=>busy,
			Error=>,
			ErrorID=>,);
			IF fbNodeGetHandle.Done THEN
			state := 2;
			END_IF
			
		2:
			fbReadVariable(
				Execute:= FALSE, 
				ConnectionHdl:= ConnectionHdl, 
				NodeHdl:= NodeHdl, 
				stNodeAddInfo:= , 
				pVariable:= pSensorValue, 
				cbData:= VariableSize, 
				Timeout:= DEFAULT_ADS_TIMEOUT, 
				Done=> , 
				Busy=> , 
				Error=> , 
				ErrorID=> , 
				cbData_R=>cbDataR );
				state := 3;
				error :=FALSE;
				
		3:		fbReadVariable(
				Execute:= TRUE, 
				ConnectionHdl:= ConnectionHdl, 
				NodeHdl:= NodeHdl, 
				stNodeAddInfo:=, 
				pVariable:= pSensorValue, 
				cbData:= VariableSize, 
				Timeout:= DEFAULT_ADS_TIMEOUT, 
				Done=>, 
				Busy=>, 
				Error=>error, 
				ErrorID=>, 
				cbData_R=>cbDataR );
				IF fbReadVariable.Done THEN
					state		:= 2;
					execute		:= FALSE;
					done		:= TRUE;
					busy		:= FALSE;
				END_IF		
		
	END_CASE
ELSE
	state := -1;
END_IF

END_FUNCTION_BLOCK

// ---- POUs/OPC Client/FB_WriteVariableOnce.TcPOU
FUNCTION_BLOCK FB_WriteVariableOnce
VAR_INPUT
	IdentifierWrite: STRING;
	NamespaceIndex: UINT;
	ConnectionHdl: DWORD;
	execute: BOOL;
	MeasuredPosition: LREAL;
END_VAR
VAR_OUTPUT
	done: BOOL;
	busy: BOOL;
	error: BOOL;
END_VAR
VAR
	/// FBs
	fbWriteVariable: UA_Write;
	fbNodeGetHandle: UA_NodeGetHandle;
	fbNodeReleaseHandle: UA_NodeReleaseHandle;
	/// Variables
	state: INT := -1;
	pMeasuredPosition: POINTER TO LREAL;
	VariableSize: UDINT;
	NodeHdl: DWORD;
	Timeout: TIME := DEFAULT_ADS_TIMEOUT;
	SesionNodeID: ST_UANodeID;
END_VAR

IF execute THEN
	CASE state OF
		
		-1:	SesionNodeID.nNamespaceIndex    			:= Namespaceindex;
			SesionNodeID.eIdentifierType				:= 1;
			SesionNodeID.sIdentifier					:= IdentifierWrite;
			VariableSize 								:= SIZEOF (LREAL);
			pMeasuredPosition							:= ADR(MeasuredPosition);
			
			
			done := FALSE;
			state:=0;
		
	    0: fbNodeGetHandle(
			Execute:=FALSE,
			ConnectionHdl:=ConnectionHdl,
			NodeID:=SesionNodeID,
			Timeout:=Timeout,
			NodeHdl=>NodeHdl,
			Done=>,
			Busy=>,
			Error=>,
			ErrorID=>,);
			state:=1;
			
		1:fbNodeGetHandle(
			Execute:=TRUE,
			ConnectionHdl:=ConnectionHdl,
			NodeID:=SesionNodeID,
			Timeout:=Timeout,
			NodeHdl=>NodeHdl,
			Done=>,
			Busy=>,
			Error=>,
			ErrorID=>,);
			IF fbNodeGetHandle.Done THEN
			state := 2;
			END_IF
			
		
				
		2: fbWriteVariable(
				Execute:=FALSE , 
				ConnectionHdl:=ConnectionHdl , 
				NodeHdl:=NodeHdl , 
				stNodeAddInfo:= , 
				pVariable:= pMeasuredPosition, 
				cbData:= VariableSize, 
				Timeout:=Timeout , 
				Done=> , 
				Busy=> , 
				Error=> , 
				ErrorID=> );
				
				state:=3;
				
		3: fbWriteVariable(
				Execute:=TRUE , 
				ConnectionHdl:=ConnectionHdl , 
				NodeHdl:=NodeHdl , 
				stNodeAddInfo:= , 
				pVariable:= pMeasuredPosition, 
				cbData:= VariableSize, 
				Timeout:=Timeout , 
				Done=> , 
				Busy=> , 
				Error=> , 
				ErrorID=> );
				IF fbWriteVariable.Done THEN
					state := 4;
				END_IF
				IF fbWriteVariable.Error THEN
					state := -1;
				END_IF
				
				
		4:		fbNodeReleaseHandle(
						Execute:= FALSE, 
						ConnectionHdl:= , 
						NodeHdl:= , 
						Timeout:= , 
						Done=> , 
						Busy=> , 
						Error=> , 
						ErrorID=> );
				state := 5;
		5: 		fbNodeReleaseHandle(
								Execute:= TRUE, 
								ConnectionHdl:= ConnectionHdl, 
								NodeHdl:= NodeHdl, 
								Timeout:= Timeout, 
								Done=> , 
								Busy=> , 
								Error=> , 
								ErrorID=> );
				IF fbNodeReleaseHandle.Done THEN
					state		:= -1;
					execute		:= FALSE;
					done		:= TRUE;
					busy		:= FALSE;
				END_IF		
	END_CASE
ELSE
	state := -1;
END_IF

END_FUNCTION_BLOCK

// ---- POUs/CAHandle/Kurvenscheibe/Powerall.TcPOU
PROGRAM Powerall
VAR
	Powerall : FB_PowerAll;
END_VAR

Powerall(enable := True);

END_PROGRAM

// ---- POUs/CAHandle/FB_PowerAll.TcPOU
FUNCTION_BLOCK FB_PowerAll
VAR_INPUT
	enable: BOOL;
	axes: ARRAY[1..axcnt] OF BOOL;
END_VAR
VAR_OUTPUT
	ison: BOOL;
END_VAR
VAR
	FBPower: ARRAY[1..axcnt] OF MC_power;
	i: UINT;
END_VAR


ison := TRUE;

FOR i:=1 TO axcnt DO
	FBPower[i](Axis:=ax[i],
		Enable			:= axes[i],
		Enable_Positive	:= enable,
		Enable_Negative	:= enable
	(*	Status			:	BOOL;	(* B *)
		Busy			: 	BOOL;	(* V *)
		Active			: 	BOOL;	(* V *)
		Valid			: 	BOOL;*)	(* E *)	(* not implemented - use Busy 
		Error			:	BOOL;	(* B *)
		ErrorID			:	UDINT;	(* E *)*)
		);
	IF (FBPower[i].Error OR ( NOT FBPower[i].Status AND axes[i]) )THEN
		ison := FALSE;
	END_IF
END_FOR
FOR i:=1 TO grpcnt DO
	FBPower[i](Axis:=grp[i],
		Enable			:= enable,
		Enable_Positive	:= enable,
		Enable_Negative	:= enable
	(*	Status			:	BOOL;	(* B *)
		Busy			: 	BOOL;	(* V *)
		Active			: 	BOOL;	(* V *)
		Valid			: 	BOOL;*)	(* E *)	(* not implemented - use Busy 
		Error			:	BOOL;	(* B *)
		ErrorID			:	UDINT;	(* E *)*)
		);
	IF (FBPower[i].Error OR NOT FBPower[i].Status) THEN
		ison := FALSE;
	END_IF
END_FOR

END_FUNCTION_BLOCK

// ---- POUs/MAIN.TcPOU
PROGRAM MAIN
VAR
	fbSkillHandleAll	: FB_SkillHandleAll;
	fbCaHandle			: FB_CAHandle;
	fbSimuLampHandle	: FB_SimuLampHandle;
	fbTranslate			: FB_TranslateInterface;
	fbTest1				: FB_TEST1;
	fbTest2				: FB_TEST2;
	fbTest3				: FB_TEST3;
	fbXInitTest			: Fb_Test_init_x;
	fbYInitTest			: Fb_Test_init_y;
	fbZInitTest			: Fb_Test_init_z;
	fbResetXTS			: Fb_ResetXTS;
	fbXInitCreme1		: Fb_Test_init_Creme1;
	fbXInitCocktail		: Fb_Test_init_Cocktail;
	fbXInitCookie		: Fb_Test_init_Cookie;
	shortTest2001		: FB_SHortTEST1;
	shortTest2002		: FB_SHortTEST2;
	shortTest2003		: FB_SHortTEST3;
	fb2001Cocktail		: FB_2001_cocktail;
	fb2002Cookie		: FB_2002cookie;
	fb2003cookie		: FB_2003_cookie;
	warmuptimer			: TON;
	warmup				: BOOL;
	i: INT;
END_VAR



fbCaHandle();
fbSkillHandleAll();
fbTranslate();
fbSimuLampHandle();
fbTest1();
fbTest2();
fbTest3();
fbxInitTest();
fbYInitTest();
fbZInitTest();
fbXInitCreme1();
fbXInitCocktail();
fbXInitCookie();
fbResetXTS();
fb2001Cocktail();
fb2002Cookie();
fb2003cookie();
warmuptimer(IN := TRUE, PT := T#55M);
IF warmuptimer.Q THEN 
	warmup := FALSE;
	warmuptimer(IN := FALSE);
END_IF
shortTest2001(execute := Maintenance);
shortTest2002(execute := ,);
shortTest2003(execute := ,);

IF ResetXTS THEN
	fbResetXTS.execute := TRUE;
END_IF
IF Restart AND restartstate = 0THEN 
	restartstate := 1;
	FOR i := 1 TO Grpcnt DO
	Moverinfo[i].blocked := FALSE;
	Moverinfo[i].reserved := FALSE;
	Moverinfo[i].surpressed := FALSE;
	Moverinfo[i].SurpressedPosition := 0;
	Moverinfo[i].nocurvestop := FALSE;
	Moverinfo[i].postposition := F_SetInSection(MoverInterface[i].Setpos + WaySectionGap);
	Moverinfo[i].preposition :=  F_SetInSection(MoverInterface[i].Setpos - WaySectionGap);
	freevelo := 300;		
	END_FOR
	restartstate := 2;
	
END_IF
IF restartstate = 4 THEN
	restart := FALSE;
	restartstate := 0;
END_IF


IF fbCaHandle.initdone THEN
fbSkillHandleAll.execute := TRUE;
fbSimuLampHandle.execute := TRUE;
ELSE
	IF fbCaHandle.cadone THEN
		fbSkillHandleAll.startinit := TRUE;
	END_IF
END_IF

END_PROGRAM

// ---- POUs/SkillHandle/FB_SkillHandleAll.TcPOU
FUNCTION_BLOCK FB_SkillHandleAll
VAR_INPUT
	execute: BOOL;
	startinit: BOOL;
END_VAR
VAR_OUTPUT
	initdone: BOOL;
END_VAR
VAR
	///FBs
	fbCalculateWaysection: FB_CalculateWaysection;
	fbCheckWaysection: FB_CheckWaysection;
	SkillHandle: ARRAY[1..grpcnt] OF FB_SkillHandle;
	freeSlotHandle: FB_FreeSlotHandle;
	i: INT;
END_VAR

IF execute THEN
	
 			FOR i:=1 TO grpcnt DO
			
			IF NOT MoverInfo[i].blocked THEN
				MoverInterface[i].Buddyenable := FALSE;
			END_IF
			 SkillHandle[i](Input:= ModuleInterface.Module[i].Input , Output=> ModuleInterface.Module[i].Output);
			 SkillAx[i] := SkillHandle[i].mymover;
			END_FOR 
			freeSlotHandle();
END_IF

IF startinit THEN
			//init auf XTS Setzen
			initdone := FALSE;
			MoverInterface[1].Targetpos := MoverInterface[1].Setpos;
			MoverInfo[1].preposition 	:= F_SetInSection(MoverInterface[1].Targetpos - WaySectionGap);
			MoverInfo[1].postposition 	:= F_SetInSection(MoverInterface[1].Targetpos + WaySectionGap);
			MoverInterface[1].Clockwise := TRUE;
			
			MoverInterface[2].Targetpos	:= MoverInterface[2].Setpos;
			MoverInfo[2].preposition 	:= F_SetInSection(MoverInterface[2].Targetpos-WaySectionGap);
			MoverInfo[2].postposition 	:= F_SetInSection(MoverInterface[2].Targetpos+WaySectionGap);
			MoverInterface[2].Clockwise := TRUE;
			
			MoverInterface[3].Targetpos	:= MoverInterface[3].Setpos;
			MoverInfo[3].preposition 	:= F_SetInSection(MoverInterface[3].Setpos - WaySectionGap);
			MoverInfo[3].postposition 	:= F_SetInSection(MoverInterface[3].Setpos + WaySectionGap);
			MoverInterface[3].Clockwise := TRUE;
			
			
			
			initdone := TRUE;
			
			FOR i := 1 TO grpcnt DO
				
				IF NOT MoverInterface[i].MovementDone THEN
					initdone := FALSE;
					
				END_IF
			END_FOR
			startinit := NOT (initdone);
			
			AwaitingAxisCnt				:= grpcnt;
END_IF

END_FUNCTION_BLOCK

// ---- POUs/SkillHandle/FB_CalculateWaysection.TcPOU
FUNCTION_BLOCK FB_CalculateWaysection
VAR_INPUT
	Clockwise: BOOL := TRUE;
	Startpos: LREAL;
	Endpos: LREAL;
	WaySectionGap: LREAL;
	Execute: BOOL;
END_VAR
VAR_OUTPUT
	Prepos: LREAL;
	Postpos: LREAL;
	done: BOOL;
END_VAR
VAR
	state: INT := 0;
	distance: LREAL;
	conflict: BOOL;
END_VAR

//DIESER FB Berechnet die waysection abhängig von start und endpos, sowie dem geünschten sicherheitsgap und der richtung
//er gibt werte zwischen 0.0 und 4000.0 aus
IF Execute THEN
	

	done := FALSE;

	CASE state OF
	0: 	conflict := FALSE;
		Prepos := 0;
		Postpos := 0;		
		state := 1;

	1:	//Überprüfung Überrundung
		IF Endpos>Startpos THEN
			distance := Endpos-Startpos;
		ELSE
			distance := Endpos + 4000 - startpos;
		END_IF
		state := 2;
	2: 
		IF Clockwise THEN
			IF ((4000.0-distance)<=(2*WaySectionGap)) THEN
				conflict := TRUE;
				//im Uhrzeigersinn
					Prepos 	:= Startpos - WaySectionGap;
					Postpos := Startpos - WaySectionGap-0.001;
					IF Prepos < 0 THEN
						Prepos := Prepos +4000.0;
					END_IF
					IF Postpos < 0 THEN
					Postpos := Postpos +4000.0;
					END_IF
					state := 100;
			ELSE //alles in ordnung
				state := 5;						
			END_IF
		ELSE
			IF ((distance)<=(2*WaySectionGap)) THEN
				conflict := TRUE;//gegen unzeigersinn
							Prepos 	:= Endpos	- WaySectionGap;
							Postpos := Endpos	- WaySectionGap - 0.001;
							IF Prepos < 0 THEN
								Prepos := Prepos +4000.0;
							END_IF
							IF Postpos < 0 THEN
								Postpos := Postpos +4000.0;
							END_IF
							IF Postpos > 4000.0 THEN
								Postpos := Postpos -4000.0;
							END_IF
							state := 100;
			ELSE //alles in ordnung
				state := 5;				
			END_IF
		END_IF
	
	
	
	
	5: 
		IF Clockwise THEN // ziel liegt im uhrzeigersinn nicht über null
		state := 10;
		ELSE
		state := 20;
		END_IF
	
	
	10: //im Uhrzeigersinn
		Prepos 	:= Startpos - WaySectionGap;
		Postpos := Endpos	+ WaySectionGap;
		IF Prepos < 0 THEN
			Prepos := Prepos +4000.0;
		END_IF
		IF Postpos > 4000.0 THEN
			Postpos := Postpos -4000.0;
		END_IF
		state := 100;
	
		
	20://gegen Uhrzeigersinn
		Prepos 	:= Endpos	- WaySectionGap;
		Postpos := Startpos + WaySectionGap;
		IF Prepos < 0 THEN
			Prepos := Prepos +4000.0;
		END_IF
		IF Postpos > 4000.0 THEN
			Postpos := Postpos -4000.0;
		END_IF
		state := 100;
	
		
	100: done := TRUE;
		 execute := FALSE;
		 state := 1;
	END_CASE
ELSE state := 1;

END_IF

END_FUNCTION_BLOCK

// ---- POUs/SkillHandle/FB_CheckWaysection.TcPOU
FUNCTION_BLOCK FB_CheckWaysection
VAR_INPUT
	CheckPreposition: LREAL;
	CheckPostposition: LREAL;
	CheckMoverNo: INT;
	Execute: BOOL;
END_VAR
VAR_OUTPUT
	SectionFree: BOOL;
	axisblocking: ARRAY[1..GrpCnt] OF BOOL;
	done: BOOL;
	busy: BOOL;
END_VAR
VAR
	i: INT;
	state: INT := 0;
	test: INT;
END_VAR

IF Execute THEN
	busy := TRUE;
	done := FALSE;

CASE state OF
	0: //überprüfen ob checkpositionen zusammenhängend sind
		IF (CheckPreposition < CheckPostposition) THEN
			//bereich zusammenhängend:
			
		state := 10;
		ELSE state := 20;
		END_IF
		
		
	10:	//RESET VALUES
		SectionFree := TRUE;
		FOR i:=1 TO grpcnt DO
			axisblocking[i] := FALSE;
		END_FOR
		state := 11;	
	11: //checkpositionen zusammenhängend
		FOR i := 1 TO grpcnt DO
			
		IF NOT (i=CheckMoverNo) THEN
			IF MoverInfo[i].postposition>MoverInfo[i].preposition 
				THEN
				//DER RESERVIERTE BEREICH GEHT NICHT ÜBER NULL:	
					
					// gesamter bereich umschlungen?
					IF ((CheckPostposition>MoverInfo[i].postposition)AND(CheckPreposition<MoverInfo[i].preposition))
					THEN 
							SectionFree := FALSE;
							axisblocking[i] := TRUE;
							test := test +1;	
					END_IF
					// Grenze in Bereich?
					IF((CheckPostposition>=MoverInfo[i].preposition) AND (CheckPostposition<=MoverInfo[i].postposition)) OR ((CheckPreposition>=MoverInfo[i].preposition) AND (CheckPreposition<=MoverInfo[i].postposition)) 
						THEN 
							SectionFree := FALSE;
							axisblocking[i] := TRUE;
							test := test +1;	
					END_IF
				
				
				ELSE
				//DER RESERVIERTE BEREICH GEHT ÜBER NULL!
				
				//Splitten des Bereichs:
				//Bereich 1: 0 bis Postpos:
					// Grenze in Bereich?
					IF((CheckPostposition>=0.0) AND (CheckPostposition<=MoverInfo[i].postposition)) OR ((CheckPreposition>=0.0) AND (CheckPreposition<=MoverInfo[i].postposition)) 
						THEN 
							SectionFree := FALSE;
							axisblocking[i] := TRUE;
							test := test +1;	
					END_IF
				
				//Bereich 2: Prepos bis 4000
					// Grenze in Bereich?
					IF((CheckPostposition>=MoverInfo[i].preposition) AND (CheckPostposition<=raillength)) OR ((CheckPreposition>=MoverInfo[i].preposition) AND (CheckPreposition<=raillength)) 
						THEN 
							SectionFree := FALSE;
							axisblocking[i] := TRUE;
							test := test +1;	
					END_IF	
			END_IF
		END_IF		
		END_FOR
		state := 200;	
	
	
	
	
	20:	//RESET VALUES
		SectionFree := TRUE;
		FOR i:=1 TO grpcnt DO
			axisblocking[i] := FALSE;
		END_FOR
		state := 21;
	

	21: //checkpositionen NICHT zusammenhängend:
		
		//Bereich von 0 bis CheckPostpos
		FOR i := 1 TO grpcnt DO
			
			IF NOT (i=CheckMoverNo) THEN
				IF MoverInfo[i].postposition>MoverInfo[i].preposition 
					THEN
					//DER RESERVIERTE BEREICH GEHT NICHT ÜBER NULL:	
						
						// gesamter bereich umschlungen?
						IF ((CheckPostposition>MoverInfo[i].postposition)AND(0.0<MoverInfo[i].preposition))
						THEN 
								SectionFree := FALSE;
								axisblocking[i] := TRUE;
								test := test +1;	
						END_IF
						// Grenze in Bereich?
						IF((CheckPostposition>MoverInfo[i].preposition) AND (CheckPostposition<=MoverInfo[i].postposition)) OR ((0.0>=MoverInfo[i].preposition) AND (0.0<=MoverInfo[i].postposition)) 
							THEN 
								SectionFree := FALSE;
								axisblocking[i] := TRUE;
								test := test +1;	
						END_IF
					
					
					ELSE
					//DER RESERVIERTE BEREICH GEHT ÜBER NULL!
					
					//Splitten des Bereichs:
					//Bereich 1: 0 bis Postpos:
						// Grenze in Bereich?
						IF((CheckPostposition>=0.0) AND (CheckPostposition<=MoverInfo[i].postposition)) OR ((0.0>=0.0) AND (0.0<=MoverInfo[i].postposition)) 
							THEN 
								SectionFree := FALSE;
								axisblocking[i] := TRUE;
								test := test +1;	
						END_IF
					
					//Bereich 2: Prepos bis 4000
						// Grenze in Bereich?
						IF((CheckPostposition>=MoverInfo[i].preposition) AND (CheckPostposition<=raillength)) OR ((0.0>=MoverInfo[i].preposition) AND (0.0<=raillength)) 
							THEN 
								SectionFree := FALSE;
								axisblocking[i] := TRUE;
								test := test +1;	
						END_IF	
				END_IF
			END_IF		
		END_FOR
		//Bereich von CheckPrepos bis Laillenth
		FOR i := 1 TO grpcnt DO
			
		IF NOT (i=CheckMoverNo) THEN
			IF MoverInfo[i].postposition>MoverInfo[i].preposition 
				THEN
				//DER RESERVIERTE BEREICH GEHT NICHT ÜBER NULL:	
					
					// gesamter bereich umschlungen?
					IF ((Raillength>MoverInfo[i].postposition)AND(CheckPreposition<MoverInfo[i].preposition))
					THEN 
							SectionFree := FALSE;
							axisblocking[i] := TRUE;
							test := test +1;	
					END_IF
					// Grenze in Bereich?
					IF((Raillength>=MoverInfo[i].preposition) AND (Raillength<=MoverInfo[i].postposition)) OR ((CheckPreposition>=MoverInfo[i].preposition) AND (CheckPreposition<=MoverInfo[i].postposition)) 
						THEN 
							SectionFree := FALSE;
							axisblocking[i] := TRUE;
							test := test +1;	
					END_IF
				
				
				ELSE
				//DER RESERVIERTE BEREICH GEHT ÜBER NULL!
				
				//Splitten des Bereichs:
				//Bereich 1: 0 bis Postpos:
					// Grenze in Bereich?
					IF((Raillength>=0.0) AND (Raillength<=MoverInfo[i].postposition)) OR ((CheckPreposition>=0.0) AND (CheckPreposition<=MoverInfo[i].postposition)) 
						THEN 
							SectionFree := FALSE;
							axisblocking[i] := TRUE;
							test := test +1;	
					END_IF
				
				//Bereich 2: Prepos bis 4000
					// Grenze in Bereich?
					IF((Raillength>=MoverInfo[i].preposition) AND (Raillength<=raillength)) OR ((CheckPreposition>=MoverInfo[i].preposition) AND (CheckPreposition<=raillength)) 
						THEN 
							SectionFree := FALSE;
							axisblocking[i] := TRUE;
							test := test +1;	
					END_IF	
				END_IF
			END_IF		
		END_FOR
		state := 200;
	200: 
		done := TRUE;
		busy := FALSE;
		Execute := FALSE;
		state := 0;
	
END_CASE

ELSE 
state := 0;
END_IF

END_FUNCTION_BLOCK

// ---- POUs/SkillHandle/FB_SkillHandle.TcPOU
FUNCTION_BLOCK FB_SkillHandle
VAR_INPUT
	Input: DUT_MODULE_INTERFACE_INPUT;
END_VAR
VAR_OUTPUT
	Output: DUT_MODULE_INTERFACE_OUTPUT;
	mymover: INT;
END_VAR
VAR
	goon: BOOL;
	nextstate: INT;
	myTimer: TOF;
	state: INT := -10;
	MoverNo: INT := 0;
	InitMoverNo: INT := 0;
	Nextaxis: INT := 0;
	measuredcycles: INT := 0;
	///Instances:
	fbTransport: FB_Transport;
	fbSuppressedTransport: FB_Transport;
	suppressed: BOOL;
	fbAutoBlock: FB_AutoBlock;
	fbUnblockTimer: FB_AutoBlock;
	fbZTransport: FB_ZTransport;
	i: INT;
	tempposition: LREAL;
	Timeout: TON;
	IdleTimer: TON;
	curvedistance: LREAL;
	idletempposition: LREAL;
	fbIdleReservedTransport: FB_FreeTransport;
	repeatcounter	: INT;
END_VAR

mymover := MoverNo;

IF NOT restart THEN

IF (NOT (MoverNo = 0)) THEN
	IF MoverInfo[MoverNo].surpressed
		THEN	suppressed := TRUE;
		ELSE	suppressed := FALSE;
	END_IF
	IF NOT MoverInfo[MoverNo].blocked THEN
		MoverInterface[MoverNo].Buddyenable := FALSE;
	END_IF
END_IF

IF NOT MoverNo = 0 THEN
	Output.StateValue[0].Description := 'Current Velocity of current Mover';
	Output.StateValue[0].Dummy		:= FALSE;
	Output.StateValue[0].Name		:= 'Velocity';
	Output.StateValue[0].Unit		:= '[mm/s]';
	Output.StateValue[0].Value 		:= ax[2*MoverNo].NcToPlc.ActVelo;
END_IF
IF NOT suppressed THEN
	//normaler Modus, suppressed = FALSE
	CASE state OF
		
			// SKILLWERTE SCHREIBEN
			-10:
				// MODUL INITIALISIEREN
				Output.Dummy 	:= FALSE;
				Output.Name		:= 'TRANSPORTMODUL';
				Output.CurrentTaskDescription	:= 'Initializing';
				Output.ID		:= 1234; ////muss sich ändern!
				
				// SKILL 0 Calibrating 
				
				Output.SkillOutput[0].Name 	:= 'Position Calibration';
				Output.SkillOutput[0].ID 	:= 1321 ;
				Output.SkillOutput[0].Ready  := FALSE ;
				Output.SkillOutput[0].Dummy  := FALSE ;
				Output.SkillOutput[0].Done   := FALSE ; 
				Output.SkillOutput[0].Busy   := FALSE ;
				Output.SkillOutput[0].ParameterOutput[0].Name := 'StringValue: ModuleServerUrl in format opc.tcp:192.168.175.xxx:4840' ; 
				Output.SkillOutput[0].ParameterOutput[0].Dummy:= FALSE;
				Output.SkillOutput[0].ParameterOutput[0].Required:= TRUE ;
	            Output.SkillOutput[0].ParameterOutput[0].MinValue:= 0 ;
				Output.SkillOutput[0].ParameterOutput[0].MaxValue:= 0 ;
				Output.SkillOutput[0].ParameterOutput[1].Name := 'StringValue: Module Output String Identifier (Sensor) ' ; 
				Output.SkillOutput[0].ParameterOutput[1].Dummy:= FALSE;
				Output.SkillOutput[0].ParameterOutput[1].Required:= TRUE ;
	            Output.SkillOutput[0].ParameterOutput[1].MinValue:= 0 ;
				Output.SkillOutput[0].ParameterOutput[1].MaxValue:= 0 ;
				Output.SkillOutput[0].ParameterOutput[2].Name := 'StringValue: Module Input String Identifier (Position/Lreal) ' ; 
				Output.SkillOutput[0].ParameterOutput[2].Dummy:= FALSE;
				Output.SkillOutput[0].ParameterOutput[2].Required:= TRUE ;
	            Output.SkillOutput[0].ParameterOutput[2].MinValue:= 0 ;
				Output.SkillOutput[0].ParameterOutput[2].MaxValue:= 0 ;
				
				
				
				// SKILL 1 reserve INITIALISIEREN
	
				Output.SkillOutput[1].Name 	:= 'Reserve';
				Output.SkillOutput[1].ID 	:= 1310 ;
				Output.SkillOutput[1].Ready  := FALSE ;
				Output.SkillOutput[1].Dummy  := FALSE ;
				Output.SkillOutput[1].Done   := FALSE ; 
				Output.SkillOutput[1].Busy   := FALSE ;
				Output.SkillOutput[1].ParameterOutput[1].Name := 'TaskID' ; 
				Output.SkillOutput[1].ParameterOutput[1].Dummy:= FALSE;
				Output.SkillOutput[1].ParameterOutput[1].Required:= TRUE ;
	            Output.SkillOutput[1].ParameterOutput[1].MinValue:= 1 ;
				Output.SkillOutput[1].ParameterOutput[1].MaxValue:=30000 ;
				
				
			 
	            // SKILL 2 unreserve INITIALISIEREN 
	           
	            Output.SkillOutput[2].Name   :='Unreserve' ;
	            Output.SkillOutput[2].ID     := 1311 ;	
				Output.SkillOutput[2].Ready  := FALSE ;
				Output.SkillOutput[2].Dummy  := FALSE ; 
	            Output.SkillOutput[2].Done   := FALSE ;
				Output.SkillOutput[2].Busy   := FALSE ;
				Output.SkillOutput[2].ParameterOutput[1].Name := 'TaskID';
				Output.SkillOutput[2].ParameterOutput[1].Dummy:= FALSE;
				Output.SkillOutput[2].ParameterOutput[1].Required:= TRUE ;
				Output.SkillOutput[2].ParameterOutput[1].MinValue:= 1;
				Output.SkillOutput[2].ParameterOutput[1].MaxValue:=30000 ;
	             
				// SKILL 3 block INITIALISIEREN 
				
